		IF Trips_DB.Section[j].Sust.ChrgRly1FaultDelay_TON.Q = TRUE THEN 
			Trips_DB.Section[j].Sust.ChargeRelay1_FailtoClose := TRUE; 
			Trips_DB.Section[j].Sust.ChrgRly1FaultDelay_TON (IN:= FALSE);
		END_IF;
	ELSE
		Trips_DB.Section[j].Sust.ChrgRly1FaultDelay_TON (IN:= FALSE);	
	END_IF;

		//fail to open
	IF LCP.Section[j].Sust.CloseChargeRelay1 = FALSE AND LCP.Section[j].Sust.ChargeRelay1_close = TRUE THEN 
		//start timer
		Trips_DB.Section[j].Sust.ChrgRly1FaultDelay_TON (IN:= TRUE, PT := ChrgRlyFaultDelay_PT);
		
		IF Trips_DB.Section[j].Sust.ChrgRly1FaultDelay_TON.Q = TRUE THEN 
			Trips_DB.Section[j].Sust.ChargeRelay1_FailtoOpen := TRUE; 
			Trips_DB.Section[j].Sust.ChrgRly1FaultDelay_TON (IN:= FALSE);
		END_IF;
	ELSE
		Trips_DB.Section[j].Sust.ChrgRly1FaultDelay_TON (IN:= FALSE);
	END_IF;

	//Sust Charge rly2	
		//fail to close
	IF LCP.Section[j].Sust.CloseChargeRelay2 = TRUE AND LCP.Section[j].Sust.ChargeRelay2_close = FALSE THEN 
		//start timer
		Trips_DB.Section[j].Sust.ChrgRly2FaultDelay_TON (IN:= TRUE, PT := ChrgRlyFaultDelay_PT);
		
		IF Trips_DB.Section[j].Sust.ChrgRly2FaultDelay_TON.Q = TRUE THEN 
			Trips_DB.Section[j].Sust.ChargeRelay2_FailtoClose := TRUE;
			Trips_DB.Section[j].Sust.ChrgRly2FaultDelay_TON (IN:= FALSE);
		END_IF;
	ELSE
		Trips_DB.Section[j].Sust.ChrgRly2FaultDelay_TON (IN:= FALSE);
	END_IF;
	
		//fail to open
	IF LCP.Section[j].Sust.CloseChargeRelay2 = FALSE AND LCP.Section[j].Sust.ChargeRelay2_close = TRUE THEN 
		//start timer
		Trips_DB.Section[j].Sust.ChrgRly2FaultDelay_TON (IN:= TRUE, PT := ChrgRlyFaultDelay_PT);
		
		IF Trips_DB.Section[j].Sust.ChrgRly2FaultDelay_TON.Q = TRUE THEN 
			Trips_DB.Section[j].Sust.ChargeRelay2_FailtoOpen := TRUE; 
			Trips_DB.Section[j].Sust.ChrgRly2FaultDelay_TON (IN:= FALSE);
		END_IF;
	ELSE
		Trips_DB.Section[j].Sust.ChrgRly2FaultDelay_TON (IN:= FALSE);
	END_IF;

	//Sust dump rly1
		//fail to open
	IF LCP.Section[j].Sust.OpenDumpRelay1 = TRUE AND LCP.Section[j].Sust.DumpRelay1_close = TRUE THEN 
		//start timer
		Trips_DB.Section[j].Sust.DumpRly1FaultDelay_TON (IN := TRUE, PT := DumpRlyFaultDelay_PT);

		IF Trips_DB.Section[j].Sust.DumpRly1FaultDelay_TON.Q = TRUE THEN 
			Trips_DB.Section[j].Sust.DumpRelay1_FailtoOpen := TRUE; 
			Trips_DB.Section[j].Sust.DumpRly1FaultDelay_TON (IN:= FALSE);
		END_IF; 
	ELSE
		Trips_DB.Section[j].Sust.DumpRly1FaultDelay_TON (IN:= FALSE);
	END_IF;

		//fail to close
	IF LCP.Section[j].Sust.OpenDumpRelay1 = FALSE AND LCP.Section[j].Sust.DumpRelay1_close = FALSE THEN 
		//start timer
		Trips_DB.Section[j].Sust.DumpRly1FaultDelay_TON (IN := TRUE, PT := DumpRlyFaultDelay_PT); 
		
		IF Trips_DB.Section[j].Sust.DumpRly1FaultDelay_TON.Q = TRUE THEN 
			Trips_DB.Section[j].Sust.DumpRelay1_FailtoClose := TRUE; 
			Trips_DB.Section[j].Sust.DumpRly1FaultDelay_TON (IN:= FALSE);
		END_IF;
	ELSE
		Trips_DB.Section[j].Sust.DumpRly1FaultDelay_TON (IN:= FALSE);
	END_IF;

	//Sust dump rly2
		//fail to open
	IF LCP.Section[j].Sust.OpenDumpRelay2 = TRUE AND LCP.Section[j].Sust.DumpRelay2_close = TRUE THEN 
		//start timer
		Trips_DB.Section[j].Sust.DumpRly2FaultDelay_TON (IN := TRUE, PT := DumpRlyFaultDelay_PT); 
		
		IF Trips_DB.Section[j].Sust.DumpRly2FaultDelay_TON.Q = TRUE THEN 
			Trips_DB.Section[j].Sust.DumpRelay2_FailtoOpen := TRUE; 
			Trips_DB.Section[j].Sust.DumpRly2FaultDelay_TON (IN:= FALSE);
		END_IF;
	ELSE
		Trips_DB.Section[j].Sust.DumpRly2FaultDelay_TON (IN:= FALSE);
	END_IF;

		//fail to close
	IF LCP.Section[j].Sust.OpenDumpRelay2 = FALSE AND LCP.Section[j].Sust.DumpRelay2_close = FALSE THEN 
		//start timer
		Trips_DB.Section[j].Sust.DumpRly2FaultDelay_TON (IN := TRUE, PT := DumpRlyFaultDelay_PT); 
		IF Trips_DB.Section[j].Sust.DumpRly2FaultDelay_TON.Q = TRUE THEN 
			Trips_DB.Section[j].Sust.DumpRelay2_FailtoClose := TRUE; 
			Trips_DB.Section[j].Sust.DumpRly2FaultDelay_TON (IN:= FALSE);
		END_IF;
	ELSE
		Trips_DB.Section[j].Sust.DumpRly2FaultDelay_TON (IN:= FALSE);
	END_IF;
	
END_FOR;
//****************************************	
	
//Form Charge rly1
		//fail to close
IF LCP.Section[4].Form.CloseChargeRelay1 = TRUE AND LCP.Section[4].Form.ChargeRelay1_close = FALSE THEN 
		//start timer
		Trips_DB.Section[4].Form.ChrgRly1FaultDelay_TON (IN:= TRUE, PT := ChrgRlyFaultDelay_PT);
		
		IF Trips_DB.Section[4].Form.ChrgRly1FaultDelay_TON.Q = TRUE THEN 
			Trips_DB.Section[4].Form.ChargeRelay1_FailtoClose := TRUE; 
			Trips_DB.Section[4].Form.ChrgRly1FaultDelay_TON (IN:= FALSE);
		END_IF;
	ELSE
		Trips_DB.Section[4].Form.ChrgRly1FaultDelay_TON (IN:= FALSE);		
END_IF;

		//fail to open
IF LCP.Section[4].Form.CloseChargeRelay1 = FALSE AND LCP.Section[4].Form.ChargeRelay1_close = TRUE THEN 
		//start timer
		Trips_DB.Section[4].Form.ChrgRly1FaultDelay_TON (IN:= TRUE, PT := ChrgRlyFaultDelay_PT);
		
		IF Trips_DB.Section[4].Form.ChrgRly1FaultDelay_TON.Q = TRUE THEN 
			Trips_DB.Section[4].Form.ChargeRelay1_FailtoOpen := TRUE; 
			Trips_DB.Section[4].Form.ChrgRly1FaultDelay_TON (IN:= FALSE);
		END_IF;
	ELSE
		Trips_DB.Section[4].Form.ChrgRly1FaultDelay_TON (IN:= FALSE);
END_IF;

	//Form Charge rly2	
		//fail to close
IF LCP.Section[4].Form.CloseChargeRelay2 = TRUE AND LCP.Section[4].Form.ChargeRelay2_close = FALSE THEN 
		//start timer
		Trips_DB.Section[4].Form.ChrgRly2FaultDelay_TON (IN:= TRUE, PT := ChrgRlyFaultDelay_PT);
		
		IF Trips_DB.Section[4].Form.ChrgRly2FaultDelay_TON.Q = TRUE THEN 
			Trips_DB.Section[4].Form.ChargeRelay2_FailtoClose := TRUE; 
			Trips_DB.Section[4].Form.ChrgRly2FaultDelay_TON (IN:= FALSE);
		END_IF;
	ELSE
		Trips_DB.Section[4].Form.ChrgRly2FaultDelay_TON (IN:= FALSE);
END_IF;
	
		//fail to open
IF LCP.Section[4].Form.CloseChargeRelay2 = FALSE AND LCP.Section[4].Form.ChargeRelay2_close = TRUE THEN 
		//start timer
		Trips_DB.Section[4].Form.ChrgRly2FaultDelay_TON (IN:= TRUE, PT := ChrgRlyFaultDelay_PT);
		
		IF Trips_DB.Section[4].Form.ChrgRly2FaultDelay_TON.Q = TRUE THEN 
			Trips_DB.Section[4].Form.ChargeRelay2_FailtoOpen := TRUE; 
			Trips_DB.Section[4].Form.ChrgRly2FaultDelay_TON (IN:= FALSE);
		END_IF;
	ELSE
		Trips_DB.Section[4].Form.ChrgRly2FaultDelay_TON (IN:= FALSE);
END_IF;

	//Form dump rly1
		//fail to open
IF LCP.Section[4].Form.OpenDumpRelay1 = TRUE AND LCP.Section[4].Form.DumpRelay1_close = TRUE THEN 
		//start timer
		Trips_DB.Section[4].Form.DumpRly1FaultDelay_TON (IN := TRUE, PT := DumpRlyFaultDelay_PT);

		IF Trips_DB.Section[4].Form.DumpRly1FaultDelay_TON.Q = TRUE THEN 
			Trips_DB.Section[4].Form.DumpRelay1_FailtoOpen := TRUE; 
			Trips_DB.Section[4].Form.DumpRly1FaultDelay_TON (IN:= FALSE);
		END_IF; 
	ELSE
		Trips_DB.Section[4].Form.DumpRly1FaultDelay_TON (IN:= FALSE);
END_IF;

		//fail to close
IF LCP.Section[4].Form.OpenDumpRelay1 = FALSE AND LCP.Section[4].Form.DumpRelay1_close = FALSE THEN 
		//start timer
		Trips_DB.Section[4].Form.DumpRly1FaultDelay_TON (IN := TRUE, PT := DumpRlyFaultDelay_PT); 
		
		IF Trips_DB.Section[4].Form.DumpRly1FaultDelay_TON.Q = TRUE THEN 
			Trips_DB.Section[4].Form.DumpRelay1_FailtoClose := TRUE; 
			Trips_DB.Section[4].Form.DumpRly1FaultDelay_TON (IN:= FALSE);
		END_IF;
	ELSE
		Trips_DB.Section[4].Form.DumpRly1FaultDelay_TON (IN:= FALSE);
END_IF;

	//Form dump rly2
		//fail to open
IF LCP.Section[4].Form.OpenDumpRelay2 = TRUE AND LCP.Section[4].Form.DumpRelay2_close = TRUE THEN 
		//start timer
		Trips_DB.Section[4].Form.DumpRly2FaultDelay_TON (IN := TRUE, PT := DumpRlyFaultDelay_PT); 
		
		IF Trips_DB.Section[4].Form.DumpRly2FaultDelay_TON.Q = TRUE THEN 
			Trips_DB.Section[4].Form.DumpRelay2_FailtoOpen := TRUE; 
			Trips_DB.Section[4].Form.DumpRly2FaultDelay_TON (IN:= FALSE);
		END_IF;
	ELSE
		Trips_DB.Section[4].Form.DumpRly2FaultDelay_TON (IN:= FALSE);
END_IF;

		//fail to close
IF LCP.Section[4].Form.OpenDumpRelay2 = FALSE AND LCP.Section[4].Form.DumpRelay2_close = FALSE THEN 
		//start timer
		Trips_DB.Section[4].Form.DumpRly2FaultDelay_TON (IN := TRUE, PT := DumpRlyFaultDelay_PT); 
		IF Trips_DB.Section[4].Form.DumpRly2FaultDelay_TON.Q = TRUE THEN 
			Trips_DB.Section[4].Form.DumpRelay2_FailtoClose := TRUE; 
			Trips_DB.Section[4].Form.DumpRly2FaultDelay_TON (IN:= FALSE);
		END_IF;
	ELSE
		Trips_DB.Section[4].Form.DumpRly2FaultDelay_TON (IN:= FALSE);
END_IF;	

	//PreForm Charge rly
		//fail to close
IF (LCP.Section[4].Form.ClosePreFormChargeRly = TRUE AND LCP.Section[4].Form.PreFormChargeRly_close = FALSE) OR 
		(LCP.Section[4].Form.ClosePreFormChargeRly = FALSE AND LCP.Section[4].Form.PreFormChargeRly_close = TRUE) 
		THEN 
		//start timer
		Trips_DB.Section[4].Form.PreFormChrgRlyFaultDelay_TON (IN:= TRUE, PT := ChrgRlyFaultDelay_PT);
		
		IF Trips_DB.Section[4].Form.PreFormChrgRlyFaultDelay_TON.Q = TRUE THEN 
			Trips_DB.Section[4].Form.PreFormChrgRlyFailed := TRUE; 
			Trips_DB.Section[4].Form.PreFormChrgRlyFaultDelay_TON (IN:= FALSE);
		END_IF;
	ELSE
		Trips_DB.Section[4].Form.PreFormChrgRlyFaultDelay_TON (IN:= FALSE);
END_IF;

//form trigger charge 
		//fail to close
IF (LCP.Section[4].Form.CloseFormTrigChargeRly = TRUE AND LCP.Section[4].Form.FormTrigChargeRly_close = FALSE) OR 
		(LCP.Section[4].Form.CloseFormTrigChargeRly = FALSE AND LCP.Section[4].Form.FormTrigChargeRly_close = TRUE) 
		THEN 
		//start timer
		Trips_DB.Section[4].Form.FormTrigChrgRlyFaultDelay_TON (IN:= TRUE, PT := ChrgRlyFaultDelay_PT);
		
		IF Trips_DB.Section[4].Form.FormTrigChrgRlyFaultDelay_TON.Q = TRUE THEN 
			Trips_DB.Section[4].Form.FormTrigChrgRlyFailed := TRUE; 
			Trips_DB.Section[4].Form.FormTrigChrgRlyFaultDelay_TON (IN:= FALSE);
		END_IF;
	ELSE
		Trips_DB.Section[4].Form.FormTrigChrgRlyFaultDelay_TON (IN:= FALSE);
END_IF;

//preform trigger charge
		//fail to close
IF (LCP.Section[4].Form.ClosePreFormTrigChargeRly = TRUE AND LCP.Section[4].Form.PreFormTrigChargeRly_close = FALSE) OR 
		(LCP.Section[4].Form.ClosePreFormTrigChargeRly = FALSE AND LCP.Section[4].Form.PreFormTrigChargeRly_close = TRUE) 
		THEN 
		//start timer
		Trips_DB.Section[4].Form.PreFormTrigChrgRlyFaultDelay_TON (IN:= TRUE, PT := ChrgRlyFaultDelay_PT);
		
		IF Trips_DB.Section[4].Form.PreFormTrigChrgRlyFaultDelay_TON.Q = TRUE THEN 
			Trips_DB.Section[4].Form.PreFormTrigChrgRlyFailed := TRUE; 
			Trips_DB.Section[4].Form.PreFormTrigChrgRlyFaultDelay_TON (IN:= FALSE);
		END_IF;
	ELSE
		Trips_DB.Section[4].Form.PreFormTrigChrgRlyFaultDelay_TON (IN:= FALSE);
END_IF;

//preform dump
	//fail to close
IF (LCP.Section[4].Form.OpenPreFormDumpRly = TRUE AND LCP.Section[4].Form.PreFormDumpRly_close = FALSE) OR 
		(LCP.Section[4].Form.OpenPreFormDumpRly = FALSE AND LCP.Section[4].Form.PreFormDumpRly_close = TRUE) 
		THEN 
		//start timer
		Trips_DB.Section[4].Form.PreFormDumpRlyFaultDelay_TON (IN:= TRUE, PT := DumpRlyFaultDelay_PT);
		
		IF Trips_DB.Section[4].Form.PreFormDumpRlyFaultDelay_TON.Q = TRUE THEN 
			Trips_DB.Section[4].Form.PreFormDumpRlyFailed := TRUE; 
			Trips_DB.Section[4].Form.PreFormDumpRlyFaultDelay_TON (IN:= FALSE);
		END_IF;
	ELSE
		Trips_DB.Section[4].Form.PreFormDumpRlyFaultDelay_TON (IN:= FALSE);
END_IF;

//form trigger dump
	//fail to close
IF (LCP.Section[4].Form.OpenFormTrigDumpRly1 = TRUE AND LCP.Section[4].Form.FormTrigDumpRly1_close = FALSE) OR 
		(LCP.Section[4].Form.OpenFormTrigDumpRly1 = FALSE AND LCP.Section[4].Form.FormTrigDumpRly1_close = TRUE) 
		THEN 
		//start timer
		Trips_DB.Section[4].Form.FormTrigDumpRlyFaultDelay_TON (IN:= TRUE, PT := DumpRlyFaultDelay_PT);
		
		IF Trips_DB.Section[4].Form.FormTrigDumpRlyFaultDelay_TON.Q = TRUE THEN 
			Trips_DB.Section[4].Form.FormTrigDumpRly1Failed := TRUE; 
			Trips_DB.Section[4].Form.FormTrigDumpRlyFaultDelay_TON (IN:= FALSE);
		END_IF;
	ELSE
		Trips_DB.Section[4].Form.FormTrigDumpRlyFaultDelay_TON (IN:= FALSE);
END_IF;
	
//preform trigger dump
	//fail to close
IF (LCP.Section[4].Form.OpenPreFormTrigDumpRly1 = TRUE AND LCP.Section[4].Form.PreFormTrigDumpRly1_close = FALSE) OR 
		(LCP.Section[4].Form.OpenPreFormTrigDumpRly1 = FALSE AND LCP.Section[4].Form.PreFormTrigDumpRly1_close = TRUE) 
		THEN 
		//start timer
		Trips_DB.Section[4].Form.PreFormTrigDumpRlyFaultDelay_TON (IN:= TRUE, PT := DumpRlyFaultDelay_PT);
		
		IF Trips_DB.Section[4].Form.PreFormTrigDumpRlyFaultDelay_TON.Q = TRUE THEN 
			Trips_DB.Section[4].Form.PreFormTrigDumpRly1Failed := TRUE; 
			Trips_DB.Section[4].Form.PreFormTrigDumpRlyFaultDelay_TON (IN:= FALSE);
		END_IF;
	ELSE
		Trips_DB.Section[4].Form.PreFormTrigDumpRlyFaultDelay_TON (IN:= FALSE);
END_IF;
	

// if rly fail to close or fail to open then trips_db.rly_failed - for alarms	
FOR j := 1 TO 3 BY 1 DO
	//peak
	IF Trips_DB.Section[j].Peak.ChargeRelay1_FailtoClose = TRUE OR Trips_DB.Section[j].Peak.ChargeRelay1_FailtoOpen = TRUE THEN
		Trips_DB.Section[j].Peak.ChargeRelay1_Failed := TRUE;  
	END_IF;
	
	IF Trips_DB.Section[j].Peak.ChargeRelay2_FailtoClose = TRUE OR Trips_DB.Section[j].Peak.ChargeRelay2_FailtoOpen = TRUE THEN
		Trips_DB.Section[j].Peak.ChargeRelay2_Failed := TRUE;  
	END_IF;
	
	IF Trips_DB.Section[j].Peak.DumpRelay1_FailtoClose = TRUE OR Trips_DB.Section[j].Peak.DumpRelay1_FailtoOpen = TRUE THEN
		Trips_DB.Section[j].Peak.DumpRelay1_Failed := TRUE;  
	END_IF;
	
	IF Trips_DB.Section[j].Peak.DumpRelay2_FailtoClose = TRUE OR Trips_DB.Section[j].Peak.DumpRelay2_FailtoOpen = TRUE THEN
		Trips_DB.Section[j].Peak.DumpRelay2_Failed := TRUE;  
	END_IF;
	
	//sust
	IF Trips_DB.Section[j].Sust.ChargeRelay1_FailtoClose = TRUE OR Trips_DB.Section[j].Sust.ChargeRelay1_FailtoOpen = TRUE THEN
		Trips_DB.Section[j].Sust.ChargeRelay1_Failed := TRUE;  
	END_IF;
	
	IF Trips_DB.Section[j].Sust.ChargeRelay2_FailtoClose = TRUE OR Trips_DB.Section[j].Sust.ChargeRelay2_FailtoOpen = TRUE THEN
		Trips_DB.Section[j].Sust.ChargeRelay2_Failed := TRUE;  
	END_IF;
	
	IF Trips_DB.Section[j].Sust.DumpRelay1_FailtoClose = TRUE OR Trips_DB.Section[j].Sust.DumpRelay1_FailtoOpen = TRUE THEN
		Trips_DB.Section[j].Sust.DumpRelay1_Failed := TRUE;  
	END_IF;
	
	IF Trips_DB.Section[j].Sust.DumpRelay2_FailtoClose = TRUE OR Trips_DB.Section[j].Sust.DumpRelay2_FailtoOpen = TRUE THEN
		Trips_DB.Section[j].Sust.DumpRelay2_Failed := TRUE;  
	END_IF;
	
END_FOR;

//any system tripped
FOR k := 1 TO 4 BY 1 DO
	IF Trips_DB.Section[k].SystemTripped = TRUE OR Trips_DB.MCPsystemTripped = TRUE THEN
		Trips_DB.AnySystemTripped := TRUE;
		ELSE
			Trips_DB.AnySystemTripped := FALSE;
	END_IF;
END_FOR

// no faulted detected
IF (Trips_DB.AnySystemTripped = FALSE AND
	Trips_DB.AnyChargerOverTemp = FALSE AND
	Trips_DB.AnyChargerLoadFault = FALSE AND  //no charger fault is a permissives to charge
	Trips_DB.AnyChargerInterlockOpen = FALSE AND
	Trips_DB.AnyChargerFaulted = FALSE AND
	Trips_DB.AnyEstopPressed = FALSE AND
	Trips_DB.AnyDumpRlyFail = FALSE AND
	Trips_DB.AnyChargeRlyFail = FALSE AND 
	Trips_DB.AllDCpsuOK = TRUE AND
	Trips_DB.AnyLossInhibitSignal = FALSE AND
	Trips_DB.AnyLossHVONsignal = FALSE AND 
	Trips_DB.MachineGNDrlyFailed = FALSE AND 
	Trips_DB.ChargingTimerRunout = FALSE AND
	Trips_DB.ChargedTimerRunout = FALSE AND
	Trips_DB.DumpTimerRunout) OR HMI_DB.NoFaultDetectedBP = TRUE //admin bypass
	THEN
		Trips_DB.NoFaultDetected := TRUE;
	ELSE
		Trips_DB.NoFaultDetected := FALSE;
END_IF;


(*
FOR i := 1 TO 10 BY 1 DO
	IF (Trips_DB.Coil[i].ACInterlockRelayFailedtoClose = TRUE OR 
		Trips_DB.Coil[i].ACInterlockRelayFailedtoOpen = TRUE OR 
		Trips_DB.Coil[i].ChargeRelay_FailtoClose = TRUE OR
		Trips_DB.Coil[i].ChargeRelay_FailtoOpen = TRUE OR
		Trips_DB.Coil[i].DumpRelay1_FailtoClose =  TRUE OR 
		Trips_DB.Coil[i].DumpRelay1_FailtoOpen = TRUE OR 
		Trips_DB.Coil[i].DumpRelay2_FailtoClose =  TRUE OR 
		Trips_DB.Coil[i].DumpRelay2_FailtoOpen = TRUE OR 
		Trips_DB.Coil[i].ChargerVoltageReadingFaulted = TRUE OR
		Trips_DB.Coil[i].CurrentReadingFaulted = TRUE OR
		Devices.Coil[i].Local_EstopPB_Pressed = TRUE OR
		Devices.Coil[i].LossPneumaticPressure = FALSE) AND Devices.Coil[i].CoilEnabled = TRUE 	
		THEN
			Devices.Coil[i].SystemFaulted := TRUE;
	END_IF
	
	IF Devices.Coil[i].SystemFaulted = TRUE THEN
		Trips_DB.SystemTripped := TRUE;
	END_IF;
END_FOR;

//*********************************** Test
(*IF InstrumentReading.R2_01_CH01 <= 0.0 THEN
	delay2s(input := FALSE);
ELSE 
	delay2s (input := TRUE);
END_IF;
bTest := delay2s.output;
*)
// Instrumentation Hardware trip
//Input.R2_01_00_Status.0;
*)
//************** Clear System Fault
IF Trips_DB.ClearAllFaults = TRUE OR stControl.ClearAllFaults = TRUE THEN
	//Trips_DB.InstrumentationFaulted := FALSE;

	Trips_DB.MCPsystemTripped := FALSE; //reset mcp trip
	Trips_DB.AnyChargerOverTemp := FALSE;
	Trips_DB.AnyChargerLoadFault := FALSE;  
	Trips_DB.AnyChargerInterlockOpen := FALSE;
	Trips_DB.AnyChargerFaulted := FALSE;
	Trips_DB.AnyEstopPressed := FALSE;
	Trips_DB.AnyDumpRlyFail := FALSE;
	Trips_DB.AnyChargeRlyFail := FALSE;
	Trips_DB.MasterStopPBPressed := FALSE; //this is only for alarms
	Trips_DB.CageEStopCircuitBroken := FALSE;
	Trips_DB.MCPLossDCpower := FALSE;
	Trips_DB.AnyLossInhibitSignal := FALSE;
	Trips_DB.AnyLossHVONsignal := FALSE;
	Trips_DB.MachineGNDrlyFailed := FALSE;
	Trips_DB.ChargingTimerRunout := FALSE;
	Trips_DB.ChargedTimerRunout  := FALSE;
	Trips_DB.DumpTimerRunout := FALSE;
	//Trips_DB.AnyACInterlockFail := FALSE;
	//reset relay trips
	FOR j := 1 TO 3 BY 1 DO 
		//reset relay faults
		Trips_DB.Section[j].SystemTripped := FALSE;
		//Peaking
		Trips_DB.Section[j].Peak.DumpRelay1_FailtoClose := FALSE;
		Trips_DB.Section[j].Peak.DumpRelay1_FailtoOpen := FALSE;
		Trips_DB.Section[j].Peak.DumpRelay2_FailtoClose := FALSE;
		Trips_DB.Section[j].Peak.DumpRelay2_FailtoOpen := FALSE;
		Trips_DB.Section[j].Peak.ChargeRelay1_FailtoClose := FALSE;
		Trips_DB.Section[j].Peak.ChargeRelay1_FailtoOpen := FALSE;
		Trips_DB.Section[j].Peak.ChargeRelay2_FailtoClose := FALSE;
		Trips_DB.Section[j].Peak.ChargeRelay2_FailtoOpen := FALSE;
		//Sust
		Trips_DB.Section[j].Sust.DumpRelay1_FailtoClose := FALSE;
		Trips_DB.Section[j].Sust.DumpRelay1_FailtoOpen := FALSE;
		Trips_DB.Section[j].Sust.DumpRelay2_FailtoClose := FALSE;
		Trips_DB.Section[j].Sust.DumpRelay2_FailtoOpen := FALSE;
		Trips_DB.Section[j].Sust.ChargeRelay1_FailtoClose := FALSE;
		Trips_DB.Section[j].Sust.ChargeRelay1_FailtoOpen := FALSE;
		Trips_DB.Section[j].Sust.ChargeRelay2_FailtoClose := FALSE;
		Trips_DB.Section[j].Sust.ChargeRelay2_FailtoOpen := FALSE;
	
	END_FOR;
	
	//FORM
	Trips_DB.Section[4].Form.ChargeRelay1_FailtoOpen := FALSE;
	Trips_DB.Section[4].Form.ChargeRelay1_FailtoClose := FALSE;
	Trips_DB.Section[4].Form.ChargeRelay1_Failed:= FALSE;
	Trips_DB.Section[4].Form.ChargeRelay2_FailtoOpen := FALSE;
	Trips_DB.Section[4].Form.ChargeRelay2_FailtoClose := FALSE;
	Trips_DB.Section[4].Form.ChargeRelay2_Failed:= FALSE;
	
	Trips_DB.Section[4].Form.DumpRelay1_FailtoOpen := FALSE;
	Trips_DB.Section[4].Form.DumpRelay1_FailtoClose := FALSE;
	Trips_DB.Section[4].Form.DumpRelay1_Failed := FALSE;
	Trips_DB.Section[4].Form.DumpRelay2_FailtoOpen := FALSE;
	Trips_DB.Section[4].Form.DumpRelay2_FailtoClose := FALSE;
	Trips_DB.Section[4].Form.DumpRelay2_Failed := FALSE;
	
	Trips_DB.Section[4].Form.PreFormChrgRlyFailed := FALSE;
	Trips_DB.Section[4].Form.FormTrigChrgRlyFailed := FALSE;
	Trips_DB.Section[4].Form.PreFormTrigChrgRlyFailed := FALSE;
	Trips_DB.Section[4].Form.PreFormDumpRlyFailed := FALSE;
	Trips_DB.Section[4].Form.FormTrigDumpRly1Failed := FALSE;
	Trips_DB.Section[4].Form.PreFormTrigDumpRly1Failed := FALSE;
	
	Trips_DB.Section[4].SystemTripped := FALSE;
	
	evtLogger.ClearAllAlarms(0, FALSE);
	//evtLogger.ClearLoggedEvents(1);
END_IF;


IF i > 8 THEN 
	i := 1;
END_IF;

IF j > 3 THEN 
	j := 1;
END_IF;

IF k > 4 THEN 
	k := 1;
END_IF;

END_PROGRAM

// ---- POUs/Alarms.TcPOU
PROGRAM Alarms
VAR
	bWarning : BOOL;
	bConfirm : BOOL;
	alarms : ARRAY[0..431] OF Alarms_FB;
	
END_VAR

// Alarm Word 1 - MCP Alarms
//MCP Alarms

Alarms_DB.MCP.AlarmWord.0 := Trips_DB.MasterStopPBPressed;
Alarms_DB.MCP.AlarmWord.1 := Trips_DB.CageEStopCircuitBroken;
Alarms_DB.MCP.AlarmWord.2 := Trips_DB.LocalModeSelected;
Alarms_DB.MCP.AlarmWord.3 := Trips_DB.MCPLossDCpower;
Alarms_DB.MCP.AlarmWord.4 := MCP_IO.Charger[1].SummaryFaulted;
Alarms_DB.MCP.AlarmWord.5 := MCP_IO.Charger[2].SummaryFaulted;
Alarms_DB.MCP.AlarmWord.6 := MCP_IO.Charger[3].SummaryFaulted;
Alarms_DB.MCP.AlarmWord.7 := MCP_IO.Charger[4].SummaryFaulted;
Alarms_DB.MCP.AlarmWord.8 := MCP_IO.Charger[5].SummaryFaulted;
Alarms_DB.MCP.AlarmWord.9 := MCP_IO.Charger[6].SummaryFaulted;
Alarms_DB.MCP.AlarmWord.10 := MCP_IO.Charger[7].SummaryFaulted;
Alarms_DB.MCP.AlarmWord.11 := MCP_IO.Charger[8].SummaryFaulted;
Alarms_DB.MCP.AlarmWord.12 := Trips_DB.ChargedTimerRunout;
Alarms_DB.MCP.AlarmWord.13 := Trips_DB.ChargingTimerRunout;
Alarms_DB.MCP.AlarmWord.14 := Trips_DB.MCPsystemTripped;
Alarms_DB.MCP.AlarmWord.15 := Trips_DB.AnyEstopPressed;

//Alarm Word 1 msg
//IE: alarms[299](evtEntry:= Tc_Events.AlarmWord11.b4, bEvt:= gvl.test, bConfirm:= bConfirm);
alarms[0](evtEntry:= Tc_Events.AlarmWord1.b0, bEvt:= Alarms_DB.MCP.AlarmWord.0, bConfirm:= bConfirm);
alarms[1](evtEntry:= Tc_Events.AlarmWord1.b1, bEvt:= Alarms_DB.MCP.AlarmWord.1, bConfirm:= bConfirm);
alarms[2](evtEntry:= Tc_Events.AlarmWord1.b2, bEvt:= Alarms_DB.MCP.AlarmWord.2, bConfirm:= bConfirm);
alarms[3](evtEntry:= Tc_Events.AlarmWord1.b3, bEvt:= Alarms_DB.MCP.AlarmWord.3, bConfirm:= bConfirm);
alarms[4](evtEntry:= Tc_Events.AlarmWord1.b4, bEvt:= Alarms_DB.MCP.AlarmWord.4, bConfirm:= bConfirm);
alarms[5](evtEntry:= Tc_Events.AlarmWord1.b5, bEvt:= Alarms_DB.MCP.AlarmWord.5, bConfirm:= bConfirm);
alarms[6](evtEntry:= Tc_Events.AlarmWord1.b6, bEvt:= Alarms_DB.MCP.AlarmWord.6, bConfirm:= bConfirm);
alarms[7](evtEntry:= Tc_Events.AlarmWord1.b7, bEvt:= Alarms_DB.MCP.AlarmWord.7, bConfirm:= bConfirm);
alarms[8](evtEntry:= Tc_Events.AlarmWord1.b8, bEvt:= Alarms_DB.MCP.AlarmWord.8, bConfirm:= bConfirm);
alarms[9](evtEntry:= Tc_Events.AlarmWord1.b9, bEvt:= Alarms_DB.MCP.AlarmWord.9, bConfirm:= bConfirm);
alarms[0](evtEntry:= Tc_Events.AlarmWord1.b10, bEvt:= Alarms_DB.MCP.AlarmWord.10, bConfirm:= bConfirm);
alarms[11](evtEntry:= Tc_Events.AlarmWord1.b11, bEvt:= Alarms_DB.MCP.AlarmWord.11, bConfirm:= bConfirm);
alarms[12](evtEntry:= Tc_Events.AlarmWord1.b12, bEvt:= Alarms_DB.MCP.AlarmWord.12, bConfirm:= bConfirm);
alarms[13](evtEntry:= Tc_Events.AlarmWord1.b13, bEvt:= Alarms_DB.MCP.AlarmWord.13, bConfirm:= bConfirm);
alarms[14](evtEntry:= Tc_Events.AlarmWord1.b14, bEvt:= Alarms_DB.MCP.AlarmWord.14, bConfirm:= bConfirm);
alarms[15](evtEntry:= Tc_Events.AlarmWord1.b15, bEvt:= Alarms_DB.MCP.AlarmWord.15, bConfirm:= bConfirm);

// Alarm Word 2 - Section 1 Alarms
Alarms_DB.Section1.AlarmWord.0 := Trips_DB.Section[1].SystemTripped;
Alarms_DB.Section1.AlarmWord.1 := Trips_DB.Section[1].LossPneumaticPressure;
Alarms_DB.Section1.AlarmWord.2 := Trips_DB.Section[1].Peak.ChargeRelay1_Failed;
Alarms_DB.Section1.AlarmWord.3 := Trips_DB.Section[1].Peak.ChargeRelay2_Failed;
Alarms_DB.Section1.AlarmWord.4 := Trips_DB.Section[1].Peak.DumpRelay1_Failed;
Alarms_DB.Section1.AlarmWord.5 := Trips_DB.Section[1].Peak.DumpRelay2_Failed;
Alarms_DB.Section1.AlarmWord.6 := Trips_DB.Section[1].Sust.ChargeRelay1_Failed;
Alarms_DB.Section1.AlarmWord.7 := Trips_DB.Section[1].Sust.ChargeRelay2_Failed;
Alarms_DB.Section1.AlarmWord.8 := Trips_DB.Section[1].Sust.DumpRelay1_Failed;
Alarms_DB.Section1.AlarmWord.9 := Trips_DB.Section[1].Sust.DumpRelay2_Failed;
Alarms_DB.Section1.AlarmWord.10 := Trips_DB.Section[1].LossDCPower;


// Alarm Word 2 - Msg
alarms[16](evtEntry:= Tc_Events.AlarmWord2.b0, bEvt:= Alarms_DB.Section1.AlarmWord.0, bConfirm:= bConfirm);
alarms[17](evtEntry:= Tc_Events.AlarmWord2.b1, bEvt:= Alarms_DB.Section1.AlarmWord.1, bConfirm:= bConfirm);
alarms[18](evtEntry:= Tc_Events.AlarmWord2.b2, bEvt:= Alarms_DB.Section1.AlarmWord.2, bConfirm:= bConfirm);
alarms[19](evtEntry:= Tc_Events.AlarmWord2.b3, bEvt:= Alarms_DB.Section1.AlarmWord.3, bConfirm:= bConfirm);
alarms[20](evtEntry:= Tc_Events.AlarmWord2.b4, bEvt:= Alarms_DB.Section1.AlarmWord.4, bConfirm:= bConfirm);
alarms[21](evtEntry:= Tc_Events.AlarmWord2.b5, bEvt:= Alarms_DB.Section1.AlarmWord.5, bConfirm:= bConfirm);
alarms[22](evtEntry:= Tc_Events.AlarmWord2.b6, bEvt:= Alarms_DB.Section1.AlarmWord.6, bConfirm:= bConfirm);
alarms[23](evtEntry:= Tc_Events.AlarmWord2.b7, bEvt:= Alarms_DB.Section1.AlarmWord.7, bConfirm:= bConfirm);
alarms[24](evtEntry:= Tc_Events.AlarmWord2.b8, bEvt:= Alarms_DB.Section1.AlarmWord.8, bConfirm:= bConfirm);
alarms[25](evtEntry:= Tc_Events.AlarmWord2.b9, bEvt:= Alarms_DB.Section1.AlarmWord.9, bConfirm:= bConfirm);
alarms[26](evtEntry:= Tc_Events.AlarmWord2.b10, bEvt:= Alarms_DB.Section1.AlarmWord.10, bConfirm:= bConfirm);
//alarms[27] - spare
//alarms[28] - spare
//alarms[29] - spare
//alarms[30] - spare
//alarms[31] - spare


// Alarm Word 3 - Section 2 Alarms
Alarms_DB.Section2.AlarmWord.0 := Trips_DB.Section[2].SystemTripped;
Alarms_DB.Section2.AlarmWord.1 := Trips_DB.Section[2].LossPneumaticPressure;
Alarms_DB.Section2.AlarmWord.2 := Trips_DB.Section[2].Peak.ChargeRelay1_Failed;
Alarms_DB.Section2.AlarmWord.3 := Trips_DB.Section[2].Peak.ChargeRelay2_Failed;
Alarms_DB.Section2.AlarmWord.4 := Trips_DB.Section[2].Peak.DumpRelay1_Failed;
Alarms_DB.Section2.AlarmWord.5 := Trips_DB.Section[2].Peak.DumpRelay2_Failed;
Alarms_DB.Section2.AlarmWord.6 := Trips_DB.Section[2].Sust.ChargeRelay1_Failed;
Alarms_DB.Section2.AlarmWord.7 := Trips_DB.Section[2].Sust.ChargeRelay2_Failed;
Alarms_DB.Section2.AlarmWord.8 := Trips_DB.Section[2].Sust.DumpRelay1_Failed;
Alarms_DB.Section2.AlarmWord.9 := Trips_DB.Section[2].Sust.DumpRelay2_Failed;
Alarms_DB.Section2.AlarmWord.10 := Trips_DB.Section[2].LossDCPower;


// Alarm Word 3 - Msg
alarms[32](evtEntry:= Tc_Events.AlarmWord3.b0, bEvt:= Alarms_DB.Section2.AlarmWord.0, bConfirm:= bConfirm);
alarms[33](evtEntry:= Tc_Events.AlarmWord3.b1, bEvt:= Alarms_DB.Section2.AlarmWord.1, bConfirm:= bConfirm);
alarms[34](evtEntry:= Tc_Events.AlarmWord3.b2, bEvt:= Alarms_DB.Section2.AlarmWord.2, bConfirm:= bConfirm);
alarms[35](evtEntry:= Tc_Events.AlarmWord3.b3, bEvt:= Alarms_DB.Section2.AlarmWord.3, bConfirm:= bConfirm);
alarms[36](evtEntry:= Tc_Events.AlarmWord3.b4, bEvt:= Alarms_DB.Section2.AlarmWord.4, bConfirm:= bConfirm);
alarms[37](evtEntry:= Tc_Events.AlarmWord3.b5, bEvt:= Alarms_DB.Section2.AlarmWord.5, bConfirm:= bConfirm);
alarms[38](evtEntry:= Tc_Events.AlarmWord3.b6, bEvt:= Alarms_DB.Section2.AlarmWord.6, bConfirm:= bConfirm);
alarms[39](evtEntry:= Tc_Events.AlarmWord3.b7, bEvt:= Alarms_DB.Section2.AlarmWord.7, bConfirm:= bConfirm);
alarms[40](evtEntry:= Tc_Events.AlarmWord3.b8, bEvt:= Alarms_DB.Section2.AlarmWord.8, bConfirm:= bConfirm);
alarms[41](evtEntry:= Tc_Events.AlarmWord3.b9, bEvt:= Alarms_DB.Section2.AlarmWord.9, bConfirm:= bConfirm);
alarms[42](evtEntry:= Tc_Events.AlarmWord3.b10, bEvt:= Alarms_DB.Section2.AlarmWord.10, bConfirm:= bConfirm);
//alarms[43] - spare
//alarms[44] - spare
//alarms[45] - spare
//alarms[46] - spare
//alarms[47] - spare

// Alarm Word 4 - Section 3 Alarms
Alarms_DB.Section3.AlarmWord.0 := Trips_DB.Section[3].SystemTripped;
Alarms_DB.Section3.AlarmWord.1 := Trips_DB.Section[3].LossPneumaticPressure;
Alarms_DB.Section3.AlarmWord.2 := Trips_DB.Section[3].Peak.ChargeRelay1_Failed;
Alarms_DB.Section3.AlarmWord.3 := Trips_DB.Section[3].Peak.ChargeRelay2_Failed;
Alarms_DB.Section3.AlarmWord.4 := Trips_DB.Section[3].Peak.DumpRelay1_Failed;
Alarms_DB.Section3.AlarmWord.5 := Trips_DB.Section[3].Peak.DumpRelay2_Failed;
Alarms_DB.Section3.AlarmWord.6 := Trips_DB.Section[3].Sust.ChargeRelay1_Failed;
Alarms_DB.Section3.AlarmWord.7 := Trips_DB.Section[3].Sust.ChargeRelay2_Failed;
Alarms_DB.Section3.AlarmWord.8 := Trips_DB.Section[3].Sust.DumpRelay1_Failed;
Alarms_DB.Section3.AlarmWord.9 := Trips_DB.Section[3].Sust.DumpRelay2_Failed;
Alarms_DB.Section3.AlarmWord.10 := Trips_DB.Section[3].LossDCPower;


// Alarm Word 4 - Msg
alarms[48](evtEntry:= Tc_Events.AlarmWord4.b0, bEvt:= Alarms_DB.Section3.AlarmWord.0, bConfirm:= bConfirm);
alarms[49](evtEntry:= Tc_Events.AlarmWord4.b1, bEvt:= Alarms_DB.Section3.AlarmWord.1, bConfirm:= bConfirm);
alarms[50](evtEntry:= Tc_Events.AlarmWord4.b2, bEvt:= Alarms_DB.Section3.AlarmWord.2, bConfirm:= bConfirm);
alarms[51](evtEntry:= Tc_Events.AlarmWord4.b3, bEvt:= Alarms_DB.Section3.AlarmWord.3, bConfirm:= bConfirm);
alarms[52](evtEntry:= Tc_Events.AlarmWord4.b4, bEvt:= Alarms_DB.Section3.AlarmWord.4, bConfirm:= bConfirm);
alarms[53](evtEntry:= Tc_Events.AlarmWord4.b5, bEvt:= Alarms_DB.Section3.AlarmWord.5, bConfirm:= bConfirm);
alarms[54](evtEntry:= Tc_Events.AlarmWord4.b6, bEvt:= Alarms_DB.Section3.AlarmWord.6, bConfirm:= bConfirm);
alarms[55](evtEntry:= Tc_Events.AlarmWord4.b7, bEvt:= Alarms_DB.Section3.AlarmWord.7, bConfirm:= bConfirm);
alarms[56](evtEntry:= Tc_Events.AlarmWord4.b8, bEvt:= Alarms_DB.Section3.AlarmWord.8, bConfirm:= bConfirm);
alarms[57](evtEntry:= Tc_Events.AlarmWord4.b9, bEvt:= Alarms_DB.Section3.AlarmWord.9, bConfirm:= bConfirm);
alarms[58](evtEntry:= Tc_Events.AlarmWord4.b10, bEvt:= Alarms_DB.Section3.AlarmWord.10, bConfirm:= bConfirm);
//alarms[59] - spare
//alarms[60] - spare
//alarms[61] - spare
//alarms[62] - spare
//alarms[63] - spare

// Alarm Word 5 - Section 4 Alarms
Alarms_DB.Section4.AlarmWord.0 := Trips_DB.Section[4].SystemTripped;
Alarms_DB.Section4.AlarmWord.1 := Trips_DB.Section[4].LossPneumaticPressure;
Alarms_DB.Section4.AlarmWord.2 := Trips_DB.Section[4].Form.ChargeRelay1_Failed;
Alarms_DB.Section4.AlarmWord.3 := Trips_DB.Section[4].Form.ChargeRelay2_Failed;
Alarms_DB.Section4.AlarmWord.4 := Trips_DB.Section[4].Form.DumpRelay1_Failed;
Alarms_DB.Section4.AlarmWord.5 := Trips_DB.Section[4].Form.DumpRelay2_Failed;
Alarms_DB.Section4.AlarmWord.6 := Trips_DB.Section[4].Form.PreFormChrgRlyFailed;
Alarms_DB.Section4.AlarmWord.7 := Trips_DB.Section[4].Form.FormTrigChrgRlyFailed;
Alarms_DB.Section4.AlarmWord.8 := Trips_DB.Section[4].Form.PreFormTrigChrgRlyFailed;
Alarms_DB.Section4.AlarmWord.9 := Trips_DB.Section[4].Form.PreFormDumpRlyFailed;
Alarms_DB.Section4.AlarmWord.10 := Trips_DB.Section[4].Form.FormTrigDumpRly1Failed;
Alarms_DB.Section4.AlarmWord.11 := Trips_DB.Section[4].Form.PreFormTrigDumpRly1Failed;
Alarms_DB.Section4.AlarmWord.12 := Trips_DB.Section[4].LossDCPower;

// Alarm Word 5 - Msg
alarms[64](evtEntry:= Tc_Events.AlarmWord5.b0, bEvt:= Alarms_DB.Section4.AlarmWord.0, bConfirm:= bConfirm);
alarms[65](evtEntry:= Tc_Events.AlarmWord5.b1, bEvt:= Alarms_DB.Section4.AlarmWord.1, bConfirm:= bConfirm);
alarms[66](evtEntry:= Tc_Events.AlarmWord5.b2, bEvt:= Alarms_DB.Section4.AlarmWord.2, bConfirm:= bConfirm);
alarms[67](evtEntry:= Tc_Events.AlarmWord5.b3, bEvt:= Alarms_DB.Section4.AlarmWord.3, bConfirm:= bConfirm);
alarms[68](evtEntry:= Tc_Events.AlarmWord5.b4, bEvt:= Alarms_DB.Section4.AlarmWord.4, bConfirm:= bConfirm);
alarms[69](evtEntry:= Tc_Events.AlarmWord5.b5, bEvt:= Alarms_DB.Section4.AlarmWord.5, bConfirm:= bConfirm);
alarms[70](evtEntry:= Tc_Events.AlarmWord5.b6, bEvt:= Alarms_DB.Section4.AlarmWord.6, bConfirm:= bConfirm);
alarms[71](evtEntry:= Tc_Events.AlarmWord5.b7, bEvt:= Alarms_DB.Section4.AlarmWord.7, bConfirm:= bConfirm);
alarms[72](evtEntry:= Tc_Events.AlarmWord5.b8, bEvt:= Alarms_DB.Section4.AlarmWord.8, bConfirm:= bConfirm);
alarms[73](evtEntry:= Tc_Events.AlarmWord5.b9, bEvt:= Alarms_DB.Section4.AlarmWord.9, bConfirm:= bConfirm);
alarms[74](evtEntry:= Tc_Events.AlarmWord5.b10, bEvt:= Alarms_DB.Section4.AlarmWord.10, bConfirm:= bConfirm);
alarms[75](evtEntry:= Tc_Events.AlarmWord5.b10, bEvt:= Alarms_DB.Section4.AlarmWord.11, bConfirm:= bConfirm);
alarms[76](evtEntry:= Tc_Events.AlarmWord5.b10, bEvt:= Alarms_DB.Section4.AlarmWord.12, bConfirm:= bConfirm);
//alarms[77] - spare
//alarms[78] - spare
//alarms[79] - spare

// Alarm Word 6 - Alarms
Alarms_DB.AlarmWord6.AlarmWord.0:= Trips_DB.Charger[1].OverTemp;
Alarms_DB.AlarmWord6.AlarmWord.1 := Trips_DB.Charger[1].InterlockOpen;
Alarms_DB.AlarmWord6.AlarmWord.2 := Trips_DB.Charger[1].LoadFaulted;
Alarms_DB.AlarmWord6.AlarmWord.3 := Trips_DB.Charger[2].OverTemp;
Alarms_DB.AlarmWord6.AlarmWord.4 := Trips_DB.Charger[2].InterlockOpen;
Alarms_DB.AlarmWord6.AlarmWord.5 := Trips_DB.Charger[2].LoadFaulted;
Alarms_DB.AlarmWord6.AlarmWord.6 := Trips_DB.Charger[3].OverTemp;
Alarms_DB.AlarmWord6.AlarmWord.7 := Trips_DB.Charger[3].InterlockOpen;
Alarms_DB.AlarmWord6.AlarmWord.8 := Trips_DB.Charger[3].LoadFaulted;
Alarms_DB.AlarmWord6.AlarmWord.9 := Trips_DB.Charger[4].OverTemp;
Alarms_DB.AlarmWord6.AlarmWord.10 := Trips_DB.Charger[4].InterlockOpen;
Alarms_DB.AlarmWord6.AlarmWord.11 := Trips_DB.Charger[4].LoadFaulted;
Alarms_DB.AlarmWord6.AlarmWord.12 := Trips_DB.Charger[5].OverTemp;
Alarms_DB.AlarmWord6.AlarmWord.13 := Trips_DB.Charger[5].InterlockOpen;
Alarms_DB.AlarmWord6.AlarmWord.14 := Trips_DB.Charger[5].LoadFaulted;

// Alarm Word 6 - Msg
alarms[80](evtEntry:= Tc_Events.AlarmWord6.b0, bEvt:= Alarms_DB.AlarmWord6.AlarmWord.0, bConfirm:= bConfirm);
alarms[81](evtEntry:= Tc_Events.AlarmWord6.b1, bEvt:= Alarms_DB.AlarmWord6.AlarmWord.1, bConfirm:= bConfirm);
alarms[82](evtEntry:= Tc_Events.AlarmWord6.b2, bEvt:= Alarms_DB.AlarmWord6.AlarmWord.2, bConfirm:= bConfirm);
alarms[83](evtEntry:= Tc_Events.AlarmWord6.b3, bEvt:= Alarms_DB.AlarmWord6.AlarmWord.3, bConfirm:= bConfirm);
alarms[84](evtEntry:= Tc_Events.AlarmWord6.b4, bEvt:= Alarms_DB.AlarmWord6.AlarmWord.4, bConfirm:= bConfirm);
alarms[85](evtEntry:= Tc_Events.AlarmWord6.b5, bEvt:= Alarms_DB.AlarmWord6.AlarmWord.5, bConfirm:= bConfirm);
alarms[86](evtEntry:= Tc_Events.AlarmWord6.b6, bEvt:= Alarms_DB.AlarmWord6.AlarmWord.6, bConfirm:= bConfirm);
alarms[87](evtEntry:= Tc_Events.AlarmWord6.b7, bEvt:= Alarms_DB.AlarmWord6.AlarmWord.7, bConfirm:= bConfirm);
alarms[88](evtEntry:= Tc_Events.AlarmWord6.b8, bEvt:= Alarms_DB.AlarmWord6.AlarmWord.8, bConfirm:= bConfirm);
alarms[89](evtEntry:= Tc_Events.AlarmWord6.b9, bEvt:= Alarms_DB.AlarmWord6.AlarmWord.9, bConfirm:= bConfirm);
alarms[90](evtEntry:= Tc_Events.AlarmWord6.b10, bEvt:= Alarms_DB.AlarmWord6.AlarmWord.10, bConfirm:= bConfirm);
alarms[91](evtEntry:= Tc_Events.AlarmWord6.b11, bEvt:= Alarms_DB.AlarmWord6.AlarmWord.11, bConfirm:= bConfirm);
alarms[92](evtEntry:= Tc_Events.AlarmWord6.b12, bEvt:= Alarms_DB.AlarmWord6.AlarmWord.12, bConfirm:= bConfirm);
//alarms[93]
//alarms[94]
//alarms[95]

// Alarm Word 7 - Charger Alarms
Alarms_DB.AlarmWord7.AlarmWord.0 := Trips_DB.Charger[6].OverTemp;
Alarms_DB.AlarmWord7.AlarmWord.1 := Trips_DB.Charger[6].InterlockOpen;
Alarms_DB.AlarmWord7.AlarmWord.2 := Trips_DB.Charger[6].LoadFaulted;
Alarms_DB.AlarmWord7.AlarmWord.3 := Trips_DB.Charger[7].OverTemp;
Alarms_DB.AlarmWord7.AlarmWord.4 := Trips_DB.Charger[7].InterlockOpen;
Alarms_DB.AlarmWord7.AlarmWord.5 := Trips_DB.Charger[7].LoadFaulted;
Alarms_DB.AlarmWord7.AlarmWord.6 := Trips_DB.Charger[8].OverTemp;
Alarms_DB.AlarmWord7.AlarmWord.7 := Trips_DB.Charger[8].InterlockOpen;
Alarms_DB.AlarmWord7.AlarmWord.8 := Trips_DB.Charger[8].LoadFaulted;
Alarms_DB.AlarmWord7.AlarmWord.9 := Trips_DB.AnyChargerOverTemp; 
Alarms_DB.AlarmWord7.AlarmWord.10 := Trips_DB.AnyChargerLoadFault; 
Alarms_DB.AlarmWord7.AlarmWord.11 := Trips_DB.AnySystemTripped; 
Alarms_DB.AlarmWord7.AlarmWord.12 := Trips_DB.MachineGNDrlyFailed; 
Alarms_DB.AlarmWord7.AlarmWord.13 := Trips_DB.AnyChargeRlyFail; 
Alarms_DB.AlarmWord7.AlarmWord.14 := Trips_DB.AnyDumpRlyFail; 
Alarms_DB.AlarmWord7.AlarmWord.15 := Trips_DB.AnyLossInhibitSignal; 

// Alarm Word 7 - Msg
alarms[96](evtEntry:= Tc_Events.AlarmWord7.b0, bEvt:= Alarms_DB.AlarmWord7.AlarmWord.0, bConfirm:= bConfirm);
alarms[97](evtEntry:= Tc_Events.AlarmWord7.b1, bEvt:= Alarms_DB.AlarmWord7.AlarmWord.1, bConfirm:= bConfirm);
alarms[98](evtEntry:= Tc_Events.AlarmWord7.b2, bEvt:= Alarms_DB.AlarmWord7.AlarmWord.2, bConfirm:= bConfirm);
alarms[99](evtEntry:= Tc_Events.AlarmWord7.b3, bEvt:= Alarms_DB.AlarmWord7.AlarmWord.3, bConfirm:= bConfirm);
alarms[100](evtEntry:= Tc_Events.AlarmWord7.b4, bEvt:= Alarms_DB.AlarmWord7.AlarmWord.4, bConfirm:= bConfirm);
alarms[101](evtEntry:= Tc_Events.AlarmWord7.b5, bEvt:= Alarms_DB.AlarmWord7.AlarmWord.5, bConfirm:= bConfirm);
alarms[102](evtEntry:= Tc_Events.AlarmWord7.b6, bEvt:= Alarms_DB.AlarmWord7.AlarmWord.6, bConfirm:= bConfirm);
alarms[103](evtEntry:= Tc_Events.AlarmWord7.b7, bEvt:= Alarms_DB.AlarmWord7.AlarmWord.7, bConfirm:= bConfirm);
alarms[104](evtEntry:= Tc_Events.AlarmWord7.b8, bEvt:= Alarms_DB.AlarmWord7.AlarmWord.8, bConfirm:= bConfirm);
alarms[105](evtEntry:= Tc_Events.AlarmWord7.b9, bEvt:= Alarms_DB.AlarmWord7.AlarmWord.9, bConfirm:= bConfirm);
alarms[106](evtEntry:= Tc_Events.AlarmWord7.b10, bEvt:= Alarms_DB.AlarmWord7.AlarmWord.10, bConfirm:= bConfirm);
alarms[107](evtEntry:= Tc_Events.AlarmWord7.b11, bEvt:= Alarms_DB.AlarmWord7.AlarmWord.11, bConfirm:= bConfirm);
alarms[108](evtEntry:= Tc_Events.AlarmWord7.b12, bEvt:= Alarms_DB.AlarmWord7.AlarmWord.12, bConfirm:= bConfirm);
alarms[109](evtEntry:= Tc_Events.AlarmWord7.b13, bEvt:= Alarms_DB.AlarmWord7.AlarmWord.13, bConfirm:= bConfirm);
alarms[110](evtEntry:= Tc_Events.AlarmWord7.b14, bEvt:= Alarms_DB.AlarmWord7.AlarmWord.14, bConfirm:= bConfirm);
alarms[111] (evtEntry:= Tc_Events.AlarmWord7.b15, bEvt:= Alarms_DB.AlarmWord7.AlarmWord.15, bConfirm:= bConfirm);


//Alarm Word 8 
Alarms_DB.AlarmWord8.AlarmWord.0 := NOT Trips_DB.AllDCpsuOK;
Alarms_DB.AlarmWord8.AlarmWord.1 := Trips_DB.AnyChargerFaulted;
Alarms_DB.AlarmWord8.AlarmWord.2 := Trips_DB.AnyLossHVONsignal;
Alarms_DB.AlarmWord8.AlarmWord.3 := NOT Trips_DB.NoFaultDetected;
Alarms_DB.AlarmWord8.AlarmWord.4 := LCP.Section[1].Peak.ShortContact1unknown;
Alarms_DB.AlarmWord8.AlarmWord.5 := LCP.Section[1].Peak.ShortContact2unknown;
Alarms_DB.AlarmWord8.AlarmWord.6 := LCP.Section[2].Peak.ShortContact1unknown;
Alarms_DB.AlarmWord8.AlarmWord.7 := LCP.Section[2].Peak.ShortContact2unknown;
Alarms_DB.AlarmWord8.AlarmWord.8 := LCP.Section[3].Peak.ShortContact1unknown;
Alarms_DB.AlarmWord8.AlarmWord.9 := LCP.Section[3].Peak.ShortContact2unknown;
Alarms_DB.AlarmWord8.AlarmWord.10 := LCP.Section[1].Sust.ShortContact1unknown;
Alarms_DB.AlarmWord8.AlarmWord.11 := LCP.Section[1].Sust.ShortContact2unknown;
Alarms_DB.AlarmWord8.AlarmWord.12 := LCP.Section[2].Sust.ShortContact1unknown;
Alarms_DB.AlarmWord8.AlarmWord.13 := LCP.Section[2].Sust.ShortContact2unknown;
Alarms_DB.AlarmWord8.AlarmWord.14 := LCP.Section[3].Sust.ShortContact1unknown;
Alarms_DB.AlarmWord8.AlarmWord.15 := LCP.Section[3].Sust.ShortContact2unknown;

//Alarm Word 8 - msg
alarms[112](evtEntry:= Tc_Events.AlarmWord8.b0, bEvt:= Alarms_DB.AlarmWord8.AlarmWord.0, bConfirm:= bConfirm);
alarms[113](evtEntry:= Tc_Events.AlarmWord8.b1, bEvt:= Alarms_DB.AlarmWord8.AlarmWord.1, bConfirm:= bConfirm);
alarms[114](evtEntry:= Tc_Events.AlarmWord8.b2, bEvt:= Alarms_DB.AlarmWord8.AlarmWord.2, bConfirm:= bConfirm);
alarms[115](evtEntry:= Tc_Events.AlarmWord8.b3, bEvt:= Alarms_DB.AlarmWord8.AlarmWord.3, bConfirm:= bConfirm);
alarms[116](evtEntry:= Tc_Events.AlarmWord8.b4, bEvt:= Alarms_DB.AlarmWord8.AlarmWord.4, bConfirm:= bConfirm);
alarms[117](evtEntry:= Tc_Events.AlarmWord8.b5, bEvt:= Alarms_DB.AlarmWord8.AlarmWord.5, bConfirm:= bConfirm);
alarms[118](evtEntry:= Tc_Events.AlarmWord8.b6, bEvt:= Alarms_DB.AlarmWord8.AlarmWord.6, bConfirm:= bConfirm);
alarms[119](evtEntry:= Tc_Events.AlarmWord8.b7, bEvt:= Alarms_DB.AlarmWord8.AlarmWord.7, bConfirm:= bConfirm);
alarms[120](evtEntry:= Tc_Events.AlarmWord8.b8, bEvt:= Alarms_DB.AlarmWord8.AlarmWord.8, bConfirm:= bConfirm);
alarms[121](evtEntry:= Tc_Events.AlarmWord8.b9, bEvt:= Alarms_DB.AlarmWord8.AlarmWord.9, bConfirm:= bConfirm);
alarms[122](evtEntry:= Tc_Events.AlarmWord8.b10, bEvt:= Alarms_DB.AlarmWord8.AlarmWord.10, bConfirm:= bConfirm);
alarms[123](evtEntry:= Tc_Events.AlarmWord8.b11, bEvt:= Alarms_DB.AlarmWord8.AlarmWord.11, bConfirm:= bConfirm);
alarms[124](evtEntry:= Tc_Events.AlarmWord8.b12, bEvt:= Alarms_DB.AlarmWord8.AlarmWord.12, bConfirm:= bConfirm);
alarms[125](evtEntry:= Tc_Events.AlarmWord8.b13, bEvt:= Alarms_DB.AlarmWord8.AlarmWord.13, bConfirm:= bConfirm);
alarms[126](evtEntry:= Tc_Events.AlarmWord8.b14, bEvt:= Alarms_DB.AlarmWord8.AlarmWord.14, bConfirm:= bConfirm);
alarms[127] (evtEntry:= Tc_Events.AlarmWord8.b15, bEvt:= Alarms_DB.AlarmWord8.AlarmWord.15, bConfirm:= bConfirm);

//Alarm Word 9 
Alarms_DB.AlarmWord9.AlarmWord.0 := LCP.Section[4].Form.ShortContact1unknown;
Alarms_DB.AlarmWord9.AlarmWord.1 := LCP.Section[4].Form.ShortContact2unknown;
Alarms_DB.AlarmWord9.AlarmWord.2 := LCP.Section[4].Form.FormTrigShortContactUnknown;
Alarms_DB.AlarmWord9.AlarmWord.3 := LCP.Section[4].Form.PreFormTrigShortContactUnknown;
Alarms_DB.AlarmWord9.AlarmWord.4 := NOT Permissives_DB.NoShortingUnknowns;
Alarms_DB.AlarmWord9.AlarmWord.5 := NOT Permissives_DB.NoInterlockPressureLoss;
Alarms_DB.AlarmWord9.AlarmWord.6 := NOT Permissives_DB.SafetyOK;
//Alarms_DB.AlarmWord9.AlarmWord.7 := 
//Alarms_DB.AlarmWord9.AlarmWord.8 := 
//Alarms_DB.AlarmWord9.AlarmWord.9 := 
//Alarms_DB.AlarmWord9.AlarmWord.10 := 
//Alarms_DB.AlarmWord9.AlarmWord.11 := 
//Alarms_DB.AlarmWord9.AlarmWord.12 := 
//Alarms_DB.AlarmWord9.AlarmWord.13 := 
//Alarms_DB.AlarmWord9.AlarmWord.14 := 
Alarms_DB.AlarmWord9.AlarmWord.15 := Trips_DB.DumpTimerRunout;

//Alarm Word 9 - msg
alarms[112](evtEntry:= Tc_Events.AlarmWord9.b0, bEvt:= Alarms_DB.AlarmWord9.AlarmWord.0, bConfirm:= bConfirm);
alarms[113](evtEntry:= Tc_Events.AlarmWord9.b1, bEvt:= Alarms_DB.AlarmWord9.AlarmWord.1, bConfirm:= bConfirm);
alarms[114](evtEntry:= Tc_Events.AlarmWord9.b2, bEvt:= Alarms_DB.AlarmWord9.AlarmWord.2, bConfirm:= bConfirm);
alarms[115](evtEntry:= Tc_Events.AlarmWord9.b3, bEvt:= Alarms_DB.AlarmWord9.AlarmWord.3, bConfirm:= bConfirm);
alarms[116](evtEntry:= Tc_Events.AlarmWord9.b4, bEvt:= Alarms_DB.AlarmWord9.AlarmWord.4, bConfirm:= bConfirm);
alarms[117](evtEntry:= Tc_Events.AlarmWord9.b5, bEvt:= Alarms_DB.AlarmWord9.AlarmWord.5, bConfirm:= bConfirm);
alarms[118](evtEntry:= Tc_Events.AlarmWord9.b6, bEvt:= Alarms_DB.AlarmWord9.AlarmWord.6, bConfirm:= bConfirm);
//alarms[119](evtEntry:= Tc_Events.AlarmWord9.b7, bEvt:= Alarms_DB.AlarmWord9.AlarmWord.7, bConfirm:= bConfirm);
//alarms[120](evtEntry:= Tc_Events.AlarmWord9.b8, bEvt:= Alarms_DB.AlarmWord9.AlarmWord.8, bConfirm:= bConfirm);
//alarms[121](evtEntry:= Tc_Events.AlarmWord9.b9, bEvt:= Alarms_DB.AlarmWord9.AlarmWord.9, bConfirm:= bConfirm);
//alarms[122](evtEntry:= Tc_Events.AlarmWord9.b10, bEvt:= Alarms_DB.AlarmWord9.AlarmWord.10, bConfirm:= bConfirm);
//alarms[123](evtEntry:= Tc_Events.AlarmWord9.b11, bEvt:= Alarms_DB.AlarmWord9.AlarmWord.11, bConfirm:= bConfirm);
//alarms[124](evtEntry:= Tc_Events.AlarmWord9.b12, bEvt:= Alarms_DB.AlarmWord9.AlarmWord.12, bConfirm:= bConfirm);
//alarms[125](evtEntry:= Tc_Events.AlarmWord9.b13, bEvt:= Alarms_DB.AlarmWord9.AlarmWord.13, bConfirm:= bConfirm);
//alarms[126](evtEntry:= Tc_Events.AlarmWord9.b14, bEvt:= Alarms_DB.AlarmWord9.AlarmWord.14, bConfirm:= bConfirm);
alarms[127] (evtEntry:= Tc_Events.AlarmWord9.b15, bEvt:= Alarms_DB.AlarmWord9.AlarmWord.15, bConfirm:= bConfirm);

//Alarm Word 11
(* uncomment this when instrument is ready
Alarms_DB.AlarmWord_11.AlarmWord.0 := Devices.Coil1.AC_Interlock_RlyOpen;
Alarms_DB.AlarmWord_11.AlarmWord.1 := Devices.Coil2.AC_Interlock_RlyOpen;
Alarms_DB.AlarmWord_11.AlarmWord.2 := Devices.Coil3.AC_Interlock_RlyOpen;
Alarms_DB.AlarmWord_11.AlarmWord.3 := Devices.Coil4.AC_Interlock_RlyOpen;
Alarms_DB.AlarmWord_11.AlarmWord.4 := Devices.Coil5.AC_Interlock_RlyOpen;
Alarms_DB.AlarmWord_11.AlarmWord.5 := Devices.Coil6.AC_Interlock_RlyOpen;
Alarms_DB.AlarmWord_11.AlarmWord.6 := Devices.Coil7.AC_Interlock_RlyOpen;
Alarms_DB.AlarmWord_11.AlarmWord.7 := Devices.Coil8.AC_Interlock_RlyOpen;
Alarms_DB.AlarmWord_11.AlarmWord.8 := Devices.Coil9.AC_Interlock_RlyOpen;
Alarms_DB.AlarmWord_11.AlarmWord.9 := Devices.Coil10.AC_Interlock_RlyOpen;
Alarms_DB.AlarmWord_11.AlarmWord.10 := NOT Permissives.AllInterlock_Closed;
*)
//Alarm Word 11 - msg
(*alarms[160](evtEntry:= Tc_Events.AlarmWord11.b0, bEvt:= Alarms_DB.AlarmWord_11.AlarmWord.0, bConfirm:= bConfirm);
alarms[161](evtEntry:= Tc_Events.AlarmWord11.b1, bEvt:= Alarms_DB.AlarmWord_11.AlarmWord.1, bConfirm:= bConfirm);
alarms[162](evtEntry:= Tc_Events.AlarmWord11.b2, bEvt:= Alarms_DB.AlarmWord_11.AlarmWord.2, bConfirm:= bConfirm);
alarms[163](evtEntry:= Tc_Events.AlarmWord11.b3, bEvt:= Alarms_DB.AlarmWord_11.AlarmWord.3, bConfirm:= bConfirm);
alarms[164](evtEntry:= Tc_Events.AlarmWord11.b4, bEvt:= Alarms_DB.AlarmWord_11.AlarmWord.4, bConfirm:= bConfirm);
alarms[165](evtEntry:= Tc_Events.AlarmWord11.b5, bEvt:= Alarms_DB.AlarmWord_11.AlarmWord.5, bConfirm:= bConfirm);
alarms[166](evtEntry:= Tc_Events.AlarmWord11.b6, bEvt:= Alarms_DB.AlarmWord_11.AlarmWord.6, bConfirm:= bConfirm);
alarms[167](evtEntry:= Tc_Events.AlarmWord11.b7, bEvt:= Alarms_DB.AlarmWord_11.AlarmWord.7, bConfirm:= bConfirm);
alarms[168](evtEntry:= Tc_Events.AlarmWord11.b8, bEvt:= Alarms_DB.AlarmWord_11.AlarmWord.8, bConfirm:= bConfirm);
alarms[169](evtEntry:= Tc_Events.AlarmWord11.b9, bEvt:= Alarms_DB.AlarmWord_11.AlarmWord.9, bConfirm:= bConfirm);
alarms[170](evtEntry:= Tc_Events.AlarmWord11.b10, bEvt:= Alarms_DB.AlarmWord_11.AlarmWord.10, bConfirm:= bConfirm);

//Alarm Word 12




//Alarm Word 22
//uncomment this when instrument is ready - commented out for testing only
Alarms_DB.AlarmWord_22.AlarmWord.0 := MCP_IO.MasterStopPB_Pressed; //NC
(*//Alarms_DB1.AlarmWord_22.AlarmWord.1 := Devices.Coil[1].Local_EstopPB_Pressed; //NC
Alarms_DB1.AlarmWord_22.AlarmWord.2 := Devices.Coil2.Local_EstopPB_Pressed; //NC
Alarms_DB1.AlarmWord_22.AlarmWord.3 := Devices.Coil3.Local_EstopPB_Pressed; //NC
Alarms_DB1.AlarmWord_22.AlarmWord.4 := Devices.Coil4.Local_EstopPB_Pressed; //NC
Alarms_DB1.AlarmWord_22.AlarmWord.5 := Devices.Coil5.Local_EstopPB_Pressed; //NC
Alarms_DB1.AlarmWord_22.AlarmWord.6 := Devices.Coil6.Local_EstopPB_Pressed; //NC
Alarms_DB1.AlarmWord_22.AlarmWord.7 := Devices.Coil7.Local_EstopPB_Pressed; //NC
Alarms_DB1.AlarmWord_22.AlarmWord.8 := Devices.Coil8.Local_EstopPB_Pressed; //NC
Alarms_DB1.AlarmWord_22.AlarmWord.9 := Devices.Coil9.Local_EstopPB_Pressed; //NC
Alarms_DB1.AlarmWord_22.AlarmWord.10 := Devices.Coil10.Local_EstopPB_Pressed; //NC
//Alarms_DB1.AlarmWord_22.AlarmWord.11 := NOT Input.R1_01_02; //0 = Manual Mode , 1 = Auto mode
//Alarms_DB1.AlarmWord_22.AlarmWord.12 := NOT Input.R1_01_01; //0 = circuit broken , 1 = circuit ok
//Alarms_DB1.AlarmWord_22.AlarmWord.13 := Spare
//Alarms_DB1.AlarmWord_22.AlarmWord.14 := Spare
//Alarms_DB1.AlarmWord_22.AlarmWord.15 := Spare
*)

//Alarm Word 22 msg
alarms[336](evtEntry:= Tc_Events.AlarmWord22.b0, bEvt:= Alarms_DB.AlarmWord_22.AlarmWord.0, bConfirm:= bConfirm);
alarms[337](evtEntry:= Tc_Events.AlarmWord22.b1, bEvt:= Alarms_DB.AlarmWord_22.AlarmWord.1, bConfirm:= bConfirm);
alarms[338](evtEntry:= Tc_Events.AlarmWord22.b2, bEvt:= Alarms_DB.AlarmWord_22.AlarmWord.2, bConfirm:= bConfirm);
alarms[339](evtEntry:= Tc_Events.AlarmWord22.b3, bEvt:= Alarms_DB.AlarmWord_22.AlarmWord.3, bConfirm:= bConfirm);
alarms[340](evtEntry:= Tc_Events.AlarmWord22.b4, bEvt:= Alarms_DB.AlarmWord_22.AlarmWord.4, bConfirm:= bConfirm);
alarms[341](evtEntry:= Tc_Events.AlarmWord22.b5, bEvt:= Alarms_DB.AlarmWord_22.AlarmWord.5, bConfirm:= bConfirm);
alarms[342](evtEntry:= Tc_Events.AlarmWord22.b6, bEvt:= Alarms_DB.AlarmWord_22.AlarmWord.6, bConfirm:= bConfirm);
alarms[343](evtEntry:= Tc_Events.AlarmWord22.b7, bEvt:= Alarms_DB.AlarmWord_22.AlarmWord.7, bConfirm:= bConfirm);
alarms[344](evtEntry:= Tc_Events.AlarmWord22.b8, bEvt:= Alarms_DB.AlarmWord_22.AlarmWord.8, bConfirm:= bConfirm);
alarms[345](evtEntry:= Tc_Events.AlarmWord22.b9, bEvt:= Alarms_DB.AlarmWord_22.AlarmWord.9, bConfirm:= bConfirm);
alarms[346](evtEntry:= Tc_Events.AlarmWord22.b10, bEvt:= Alarms_DB.AlarmWord_22.AlarmWord.10, bConfirm:= bConfirm);
alarms[347](evtEntry:= Tc_Events.AlarmWord22.b11, bEvt:= Alarms_DB.AlarmWord_22.AlarmWord.11, bConfirm:= bConfirm);
alarms[348](evtEntry:= Tc_Events.AlarmWord22.b12, bEvt:= Alarms_DB.AlarmWord_22.AlarmWord.12, bConfirm:= bConfirm);

//Alarm Word 23
(* uncomment when instrument is ready
Alarms_DB.AlarmWord_23.AlarmWord.0 := Trips_DB.Coil[1].ChargeRelay_FailtoClose; 
Alarms_DB.AlarmWord_23.AlarmWord.1 := Trips_DB.Coil[1].ChargeRelay_FailtoOpen;
Alarms_DB.AlarmWord_23.AlarmWord.2 := Trips_DB.Coil[2].ChargeRelay_FailtoClose;
Alarms_DB.AlarmWord_23.AlarmWord.3 := Trips_DB.Coil[2].ChargeRelay_FailtoOpen;
Alarms_DB.AlarmWord_23.AlarmWord.4 := Trips_DB.Coil[3].ChargeRelay_FailtoClose;
Alarms_DB.AlarmWord_23.AlarmWord.5 := Trips_DB.Coil[3].ChargeRelay_FailtoOpen;
Alarms_DB.AlarmWord_23.AlarmWord.6 := Trips_DB.Coil[4].ChargeRelay_FailtoClose;
Alarms_DB.AlarmWord_23.AlarmWord.7 := Trips_DB.Coil[4].ChargeRelay_FailtoOpen;
Alarms_DB.AlarmWord_23.AlarmWord.8 := Trips_DB.Coil[5].ChargeRelay_FailtoClose;
Alarms_DB.AlarmWord_23.AlarmWord.9 := Trips_DB.Coil[5].ChargeRelay_FailtoOpen;
Alarms_DB.AlarmWord_23.AlarmWord.10 := Trips_DB.Coil[6].ChargeRelay_FailtoClose;
Alarms_DB.AlarmWord_23.AlarmWord.11 := Trips_DB.Coil[6].ChargeRelay_FailtoOpen;
Alarms_DB.AlarmWord_23.AlarmWord.12 := Trips_DB.Coil[7].ChargeRelay_FailtoClose;
Alarms_DB.AlarmWord_23.AlarmWord.13 := Trips_DB.Coil[7].ChargeRelay_FailtoOpen;
Alarms_DB.AlarmWord_23.AlarmWord.14 := Trips_DB.Coil[8].ChargeRelay_FailtoClose;
Alarms_DB.AlarmWord_23.AlarmWord.15 := Trips_DB.Coil[9].ChargeRelay_FailtoOpen;
*)
//Alarm Word 23 msg
alarms[352](evtEntry:= Tc_Events.AlarmWord23.b0, bEvt:= Alarms_DB.AlarmWord_23.AlarmWord.0, bConfirm:= bConfirm);
alarms[353](evtEntry:= Tc_Events.AlarmWord23.b1, bEvt:= Alarms_DB.AlarmWord_23.AlarmWord.1, bConfirm:= bConfirm);
alarms[354](evtEntry:= Tc_Events.AlarmWord23.b2, bEvt:= Alarms_DB.AlarmWord_23.AlarmWord.2, bConfirm:= bConfirm);
alarms[355](evtEntry:= Tc_Events.AlarmWord23.b3, bEvt:= Alarms_DB.AlarmWord_23.AlarmWord.3, bConfirm:= bConfirm);
alarms[356](evtEntry:= Tc_Events.AlarmWord23.b4, bEvt:= Alarms_DB.AlarmWord_23.AlarmWord.4, bConfirm:= bConfirm);
alarms[357](evtEntry:= Tc_Events.AlarmWord23.b5, bEvt:= Alarms_DB.AlarmWord_23.AlarmWord.5, bConfirm:= bConfirm);
alarms[358](evtEntry:= Tc_Events.AlarmWord23.b6, bEvt:= Alarms_DB.AlarmWord_23.AlarmWord.6, bConfirm:= bConfirm);
alarms[359](evtEntry:= Tc_Events.AlarmWord23.b7, bEvt:= Alarms_DB.AlarmWord_23.AlarmWord.7, bConfirm:= bConfirm);
alarms[360](evtEntry:= Tc_Events.AlarmWord23.b8, bEvt:= Alarms_DB.AlarmWord_23.AlarmWord.8, bConfirm:= bConfirm);
alarms[361](evtEntry:= Tc_Events.AlarmWord23.b9, bEvt:= Alarms_DB.AlarmWord_23.AlarmWord.9, bConfirm:= bConfirm);
alarms[362](evtEntry:= Tc_Events.AlarmWord23.b10, bEvt:= Alarms_DB.AlarmWord_23.AlarmWord.10, bConfirm:= bConfirm);
alarms[363](evtEntry:= Tc_Events.AlarmWord23.b11, bEvt:= Alarms_DB.AlarmWord_23.AlarmWord.11, bConfirm:= bConfirm);
alarms[364](evtEntry:= Tc_Events.AlarmWord23.b12, bEvt:= Alarms_DB.AlarmWord_23.AlarmWord.12, bConfirm:= bConfirm);
alarms[365](evtEntry:= Tc_Events.AlarmWord23.b13, bEvt:= Alarms_DB.AlarmWord_23.AlarmWord.13, bConfirm:= bConfirm);
alarms[366](evtEntry:= Tc_Events.AlarmWord23.b14, bEvt:= Alarms_DB.AlarmWord_23.AlarmWord.14, bConfirm:= bConfirm);
alarms[367](evtEntry:= Tc_Events.AlarmWord23.b15, bEvt:= Alarms_DB.AlarmWord_23.AlarmWord.15, bConfirm:= bConfirm);

//Alarm Word 24
(* uncomment when instrument is ready
Alarms_DB.AlarmWord_24.AlarmWord.0 := Trips_DB.Coil[9].ChargeRelay_FailtoClose; 
Alarms_DB.AlarmWord_24.AlarmWord.1 := Trips_DB.Coil[9].ChargeRelay_FailtoOpen;
Alarms_DB.AlarmWord_24.AlarmWord.2 := Trips_DB.Coil[10].ChargeRelay_FailtoClose;
Alarms_DB.AlarmWord_24.AlarmWord.3 := Trips_DB.Coil[10].ChargeRelay_FailtoOpen;
Alarms_DB.AlarmWord_24.AlarmWord.4 := Trips_DB.Coil[1].ACInterlockRelayFailedtoClose;
Alarms_DB.AlarmWord_24.AlarmWord.5 := Trips_DB.Coil[1].ACInterlockRelayFailedtoOpen;
Alarms_DB.AlarmWord_24.AlarmWord.6 := Trips_DB.Coil[2].ACInterlockRelayFailedtoClose;
Alarms_DB.AlarmWord_24.AlarmWord.7 := Trips_DB.Coil[2].ACInterlockRelayFailedtoOpen;
Alarms_DB.AlarmWord_24.AlarmWord.8 := Trips_DB.Coil[3].ACInterlockRelayFailedtoClose;
Alarms_DB.AlarmWord_24.AlarmWord.9 := Trips_DB.Coil[3].ACInterlockRelayFailedtoOpen;
Alarms_DB.AlarmWord_24.AlarmWord.10 := Trips_DB.Coil[4].ACInterlockRelayFailedtoClose;
Alarms_DB.AlarmWord_24.AlarmWord.11 := Trips_DB.Coil[4].ACInterlockRelayFailedtoOpen;
Alarms_DB.AlarmWord_24.AlarmWord.12 := Trips_DB.Coil[5].ACInterlockRelayFailedtoClose;
Alarms_DB.AlarmWord_24.AlarmWord.13 := Trips_DB.Coil[5].ACInterlockRelayFailedtoOpen;
Alarms_DB.AlarmWord_24.AlarmWord.14 := Trips_DB.Coil[6].ACInterlockRelayFailedtoClose;
Alarms_DB.AlarmWord_24.AlarmWord.15 := Trips_DB.Coil[6].ACInterlockRelayFailedtoOpen;
*)
//Alarm Word 24 msg
alarms[368](evtEntry:= Tc_Events.AlarmWord24.b0, bEvt:= Alarms_DB.AlarmWord_24.AlarmWord.0, bConfirm:= bConfirm);
alarms[369](evtEntry:= Tc_Events.AlarmWord24.b1, bEvt:= Alarms_DB.AlarmWord_24.AlarmWord.1, bConfirm:= bConfirm);
alarms[370](evtEntry:= Tc_Events.AlarmWord24.b2, bEvt:= Alarms_DB.AlarmWord_24.AlarmWord.2, bConfirm:= bConfirm);
alarms[371](evtEntry:= Tc_Events.AlarmWord24.b3, bEvt:= Alarms_DB.AlarmWord_24.AlarmWord.3, bConfirm:= bConfirm);
alarms[372](evtEntry:= Tc_Events.AlarmWord24.b4, bEvt:= Alarms_DB.AlarmWord_24.AlarmWord.4, bConfirm:= bConfirm);
alarms[373](evtEntry:= Tc_Events.AlarmWord24.b5, bEvt:= Alarms_DB.AlarmWord_24.AlarmWord.5, bConfirm:= bConfirm);
alarms[374](evtEntry:= Tc_Events.AlarmWord24.b6, bEvt:= Alarms_DB.AlarmWord_24.AlarmWord.6, bConfirm:= bConfirm);
alarms[375](evtEntry:= Tc_Events.AlarmWord24.b7, bEvt:= Alarms_DB.AlarmWord_24.AlarmWord.7, bConfirm:= bConfirm);
alarms[376](evtEntry:= Tc_Events.AlarmWord24.b8, bEvt:= Alarms_DB.AlarmWord_24.AlarmWord.8, bConfirm:= bConfirm);
alarms[377](evtEntry:= Tc_Events.AlarmWord24.b9, bEvt:= Alarms_DB.AlarmWord_24.AlarmWord.9, bConfirm:= bConfirm);
alarms[378](evtEntry:= Tc_Events.AlarmWord24.b10, bEvt:= Alarms_DB.AlarmWord_24.AlarmWord.10, bConfirm:= bConfirm);
alarms[379](evtEntry:= Tc_Events.AlarmWord24.b11, bEvt:= Alarms_DB.AlarmWord_24.AlarmWord.11, bConfirm:= bConfirm);
alarms[380](evtEntry:= Tc_Events.AlarmWord24.b12, bEvt:= Alarms_DB.AlarmWord_24.AlarmWord.12, bConfirm:= bConfirm);
alarms[381](evtEntry:= Tc_Events.AlarmWord24.b13, bEvt:= Alarms_DB.AlarmWord_24.AlarmWord.13, bConfirm:= bConfirm);
alarms[382](evtEntry:= Tc_Events.AlarmWord24.b14, bEvt:= Alarms_DB.AlarmWord_24.AlarmWord.14, bConfirm:= bConfirm);
alarms[383](evtEntry:= Tc_Events.AlarmWord24.b15, bEvt:= Alarms_DB.AlarmWord_24.AlarmWord.15, bConfirm:= bConfirm);

//Alarm Word 25
(* uncomment when instrument is ready
Alarms_DB.AlarmWord_25.AlarmWord.0 := Trips_DB.Coil[7].ACInterlockRelayFailedtoClose;
Alarms_DB.AlarmWord_25.AlarmWord.1 := Trips_DB.Coil[7].ACInterlockRelayFailedtoOpen;
Alarms_DB.AlarmWord_25.AlarmWord.2 := Trips_DB.Coil[8].ACInterlockRelayFailedtoClose;
Alarms_DB.AlarmWord_25.AlarmWord.3 := Trips_DB.Coil[8].ACInterlockRelayFailedtoOpen;
Alarms_DB.AlarmWord_25.AlarmWord.4 := Trips_DB.Coil[9].ACInterlockRelayFailedtoClose;
Alarms_DB.AlarmWord_25.AlarmWord.5 := Trips_DB.Coil[9].ACInterlockRelayFailedtoOpen;
Alarms_DB.AlarmWord_25.AlarmWord.6 := Trips_DB.Coil[10].ACInterlockRelayFailedtoClose;
Alarms_DB.AlarmWord_25.AlarmWord.7 := Trips_DB.Coil[10].ACInterlockRelayFailedtoOpen;
Alarms_DB.AlarmWord_25.AlarmWord.8 := Trips_DB.Coil[1].DumpRelay1_FailtoClose;
Alarms_DB.AlarmWord_25.AlarmWord.9 := Trips_DB.Coil[1].DumpRelay1_FailtoOpen;
Alarms_DB.AlarmWord_25.AlarmWord.10 := Trips_DB.Coil[2].DumpRelay1_FailtoClose;
Alarms_DB.AlarmWord_25.AlarmWord.11 := Trips_DB.Coil[2].DumpRelay1_FailtoOpen;
Alarms_DB.AlarmWord_25.AlarmWord.12 := Trips_DB.Coil[3].DumpRelay1_FailtoClose;
Alarms_DB.AlarmWord_25.AlarmWord.13 := Trips_DB.Coil[3].DumpRelay1_FailtoOpen;
Alarms_DB.AlarmWord_25.AlarmWord.14 := Trips_DB.Coil[4].DumpRelay1_FailtoClose;
Alarms_DB.AlarmWord_25.AlarmWord.15 := Trips_DB.Coil[4].DumpRelay1_FailtoOpen;
*)
//Alarm Word 25 msg
alarms[384](evtEntry:= Tc_Events.AlarmWord25.b0, bEvt:= Alarms_DB.AlarmWord_25.AlarmWord.0, bConfirm:= bConfirm);
alarms[385](evtEntry:= Tc_Events.AlarmWord25.b1, bEvt:= Alarms_DB.AlarmWord_25.AlarmWord.1, bConfirm:= bConfirm);
alarms[386](evtEntry:= Tc_Events.AlarmWord25.b2, bEvt:= Alarms_DB.AlarmWord_25.AlarmWord.2, bConfirm:= bConfirm);
alarms[387](evtEntry:= Tc_Events.AlarmWord25.b3, bEvt:= Alarms_DB.AlarmWord_25.AlarmWord.3, bConfirm:= bConfirm);
alarms[388](evtEntry:= Tc_Events.AlarmWord25.b4, bEvt:= Alarms_DB.AlarmWord_25.AlarmWord.4, bConfirm:= bConfirm);
alarms[389](evtEntry:= Tc_Events.AlarmWord25.b5, bEvt:= Alarms_DB.AlarmWord_25.AlarmWord.5, bConfirm:= bConfirm);
alarms[390](evtEntry:= Tc_Events.AlarmWord25.b6, bEvt:= Alarms_DB.AlarmWord_25.AlarmWord.6, bConfirm:= bConfirm);
alarms[391](evtEntry:= Tc_Events.AlarmWord25.b7, bEvt:= Alarms_DB.AlarmWord_25.AlarmWord.7, bConfirm:= bConfirm);
alarms[392](evtEntry:= Tc_Events.AlarmWord25.b8, bEvt:= Alarms_DB.AlarmWord_25.AlarmWord.8, bConfirm:= bConfirm);
alarms[393](evtEntry:= Tc_Events.AlarmWord25.b9, bEvt:= Alarms_DB.AlarmWord_25.AlarmWord.9, bConfirm:= bConfirm);
alarms[394](evtEntry:= Tc_Events.AlarmWord25.b10, bEvt:= Alarms_DB.AlarmWord_25.AlarmWord.10, bConfirm:= bConfirm);
alarms[395](evtEntry:= Tc_Events.AlarmWord25.b11, bEvt:= Alarms_DB.AlarmWord_25.AlarmWord.11, bConfirm:= bConfirm);
alarms[396](evtEntry:= Tc_Events.AlarmWord25.b12, bEvt:= Alarms_DB.AlarmWord_25.AlarmWord.12, bConfirm:= bConfirm);
alarms[397](evtEntry:= Tc_Events.AlarmWord25.b13, bEvt:= Alarms_DB.AlarmWord_25.AlarmWord.13, bConfirm:= bConfirm);
alarms[398](evtEntry:= Tc_Events.AlarmWord25.b14, bEvt:= Alarms_DB.AlarmWord_25.AlarmWord.14, bConfirm:= bConfirm);
alarms[399](evtEntry:= Tc_Events.AlarmWord25.b15, bEvt:= Alarms_DB.AlarmWord_25.AlarmWord.15, bConfirm:= bConfirm);

//Alarm Word 26
(* uncomment when instrument is ready
Alarms_DB.AlarmWord_26.AlarmWord.0 := Trips_DB.Coil[5].DumpRelay1_FailtoClose;
Alarms_DB.AlarmWord_26.AlarmWord.1 := Trips_DB.Coil[5].DumpRelay1_FailtoOpen;
Alarms_DB.AlarmWord_26.AlarmWord.2 := Trips_DB.Coil[6].DumpRelay1_FailtoClose;
Alarms_DB.AlarmWord_26.AlarmWord.3 := Trips_DB.Coil[6].DumpRelay1_FailtoOpen;
Alarms_DB.AlarmWord_26.AlarmWord.4 := Trips_DB.Coil[7].DumpRelay1_FailtoClose;
Alarms_DB.AlarmWord_26.AlarmWord.5 := Trips_DB.Coil[7].DumpRelay1_FailtoOpen;
Alarms_DB.AlarmWord_26.AlarmWord.6 := Trips_DB.Coil[8].DumpRelay1_FailtoClose;
Alarms_DB.AlarmWord_26.AlarmWord.7 := Trips_DB.Coil[8].DumpRelay1_FailtoOpen;
Alarms_DB.AlarmWord_26.AlarmWord.8 := Trips_DB.Coil[9].DumpRelay1_FailtoClose;
Alarms_DB.AlarmWord_26.AlarmWord.9 := Trips_DB.Coil[9].DumpRelay1_FailtoOpen;
Alarms_DB.AlarmWord_26.AlarmWord.10 := Trips_DB.Coil[10].DumpRelay1_FailtoClose;
Alarms_DB.AlarmWord_26.AlarmWord.11 := Trips_DB.Coil[10].DumpRelay1_FailtoOpen;
Alarms_DB.AlarmWord_26.AlarmWord.12 := Trips_DB.Coil[1].DumpRelay2_FailtoClose;
Alarms_DB.AlarmWord_26.AlarmWord.13 := Trips_DB.Coil[1].DumpRelay2_FailtoOpen;
Alarms_DB.AlarmWord_26.AlarmWord.14 := Trips_DB.Coil[2].DumpRelay2_FailtoClose;
Alarms_DB.AlarmWord_26.AlarmWord.15 := Trips_DB.Coil[2].DumpRelay2_FailtoOpen;
*)
//Alarm Word 26 msg
alarms[400](evtEntry:= Tc_Events.AlarmWord26.b0, bEvt:= Alarms_DB.AlarmWord_26.AlarmWord.0, bConfirm:= bConfirm);
alarms[401](evtEntry:= Tc_Events.AlarmWord26.b1, bEvt:= Alarms_DB.AlarmWord_26.AlarmWord.1, bConfirm:= bConfirm);
alarms[402](evtEntry:= Tc_Events.AlarmWord26.b2, bEvt:= Alarms_DB.AlarmWord_26.AlarmWord.2, bConfirm:= bConfirm);
alarms[403](evtEntry:= Tc_Events.AlarmWord26.b3, bEvt:= Alarms_DB.AlarmWord_26.AlarmWord.3, bConfirm:= bConfirm);
alarms[404](evtEntry:= Tc_Events.AlarmWord26.b4, bEvt:= Alarms_DB.AlarmWord_26.AlarmWord.4, bConfirm:= bConfirm);
alarms[405](evtEntry:= Tc_Events.AlarmWord26.b5, bEvt:= Alarms_DB.AlarmWord_26.AlarmWord.5, bConfirm:= bConfirm);
alarms[406](evtEntry:= Tc_Events.AlarmWord26.b6, bEvt:= Alarms_DB.AlarmWord_26.AlarmWord.6, bConfirm:= bConfirm);
alarms[407](evtEntry:= Tc_Events.AlarmWord26.b7, bEvt:= Alarms_DB.AlarmWord_26.AlarmWord.7, bConfirm:= bConfirm);
alarms[408](evtEntry:= Tc_Events.AlarmWord26.b8, bEvt:= Alarms_DB.AlarmWord_26.AlarmWord.8, bConfirm:= bConfirm);
alarms[409](evtEntry:= Tc_Events.AlarmWord26.b9, bEvt:= Alarms_DB.AlarmWord_26.AlarmWord.9, bConfirm:= bConfirm);
alarms[410](evtEntry:= Tc_Events.AlarmWord26.b10, bEvt:= Alarms_DB.AlarmWord_26.AlarmWord.10, bConfirm:= bConfirm);
alarms[411](evtEntry:= Tc_Events.AlarmWord26.b11, bEvt:= Alarms_DB.AlarmWord_26.AlarmWord.11, bConfirm:= bConfirm);
alarms[412](evtEntry:= Tc_Events.AlarmWord26.b12, bEvt:= Alarms_DB.AlarmWord_26.AlarmWord.12, bConfirm:= bConfirm);
alarms[413](evtEntry:= Tc_Events.AlarmWord26.b13, bEvt:= Alarms_DB.AlarmWord_26.AlarmWord.13, bConfirm:= bConfirm);
alarms[414](evtEntry:= Tc_Events.AlarmWord26.b14, bEvt:= Alarms_DB.AlarmWord_26.AlarmWord.14, bConfirm:= bConfirm);
alarms[415](evtEntry:= Tc_Events.AlarmWord26.b15, bEvt:= Alarms_DB.AlarmWord_26.AlarmWord.15, bConfirm:= bConfirm);

//Alarm Word 27
(* uncomment when instrument is ready
Alarms_DB.AlarmWord_27.AlarmWord.0 := Trips_DB.Coil[3].DumpRelay2_FailtoClose;
Alarms_DB.AlarmWord_27.AlarmWord.1 := Trips_DB.Coil[3].DumpRelay2_FailtoOpen;
Alarms_DB.AlarmWord_27.AlarmWord.2 := Trips_DB.Coil[4].DumpRelay2_FailtoClose;
Alarms_DB.AlarmWord_27.AlarmWord.3 := Trips_DB.Coil[4].DumpRelay2_FailtoOpen;
Alarms_DB.AlarmWord_27.AlarmWord.4 := Trips_DB.Coil[5].DumpRelay2_FailtoClose;
Alarms_DB.AlarmWord_27.AlarmWord.5 := Trips_DB.Coil[5].DumpRelay2_FailtoOpen;
Alarms_DB.AlarmWord_27.AlarmWord.6 := Trips_DB.Coil[6].DumpRelay2_FailtoClose;
Alarms_DB.AlarmWord_27.AlarmWord.7 := Trips_DB.Coil[6].DumpRelay2_FailtoOpen;
Alarms_DB.AlarmWord_27.AlarmWord.8 := Trips_DB.Coil[7].DumpRelay2_FailtoClose;
Alarms_DB.AlarmWord_27.AlarmWord.9 := Trips_DB.Coil[7].DumpRelay2_FailtoOpen;
Alarms_DB.AlarmWord_27.AlarmWord.10 := Trips_DB.Coil[8].DumpRelay2_FailtoClose;
Alarms_DB.AlarmWord_27.AlarmWord.11 := Trips_DB.Coil[8].DumpRelay2_FailtoOpen;
Alarms_DB.AlarmWord_27.AlarmWord.12:= Trips_DB.Coil[9].DumpRelay2_FailtoClose;
Alarms_DB.AlarmWord_27.AlarmWord.13 := Trips_DB.Coil[9].DumpRelay2_FailtoOpen;
Alarms_DB.AlarmWord_27.AlarmWord.14 := Trips_DB.Coil[10].DumpRelay2_FailtoClose;
Alarms_DB.AlarmWord_27.AlarmWord.15 := Trips_DB.Coil[10].DumpRelay2_FailtoOpen;
*)
//Alarm Word 27 msg
alarms[416](evtEntry:= Tc_Events.AlarmWord27.b0, bEvt:= Alarms_DB.AlarmWord_27.AlarmWord.0, bConfirm:= bConfirm);
alarms[417](evtEntry:= Tc_Events.AlarmWord27.b1, bEvt:= Alarms_DB.AlarmWord_27.AlarmWord.1, bConfirm:= bConfirm);
alarms[418](evtEntry:= Tc_Events.AlarmWord27.b2, bEvt:= Alarms_DB.AlarmWord_27.AlarmWord.2, bConfirm:= bConfirm);
alarms[419](evtEntry:= Tc_Events.AlarmWord27.b3, bEvt:= Alarms_DB.AlarmWord_27.AlarmWord.3, bConfirm:= bConfirm);
alarms[420](evtEntry:= Tc_Events.AlarmWord27.b4, bEvt:= Alarms_DB.AlarmWord_27.AlarmWord.4, bConfirm:= bConfirm);
alarms[421](evtEntry:= Tc_Events.AlarmWord27.b5, bEvt:= Alarms_DB.AlarmWord_27.AlarmWord.5, bConfirm:= bConfirm);
alarms[422](evtEntry:= Tc_Events.AlarmWord27.b6, bEvt:= Alarms_DB.AlarmWord_27.AlarmWord.6, bConfirm:= bConfirm);
alarms[423](evtEntry:= Tc_Events.AlarmWord27.b7, bEvt:= Alarms_DB.AlarmWord_27.AlarmWord.7, bConfirm:= bConfirm);
alarms[424](evtEntry:= Tc_Events.AlarmWord27.b8, bEvt:= Alarms_DB.AlarmWord_27.AlarmWord.8, bConfirm:= bConfirm);
alarms[425](evtEntry:= Tc_Events.AlarmWord27.b9, bEvt:= Alarms_DB.AlarmWord_27.AlarmWord.9, bConfirm:= bConfirm);
alarms[426](evtEntry:= Tc_Events.AlarmWord27.b10, bEvt:= Alarms_DB.AlarmWord_27.AlarmWord.10, bConfirm:= bConfirm);
alarms[427](evtEntry:= Tc_Events.AlarmWord27.b11, bEvt:= Alarms_DB.AlarmWord_27.AlarmWord.11, bConfirm:= bConfirm);
alarms[428](evtEntry:= Tc_Events.AlarmWord27.b12, bEvt:= Alarms_DB.AlarmWord_27.AlarmWord.12, bConfirm:= bConfirm);
alarms[429](evtEntry:= Tc_Events.AlarmWord27.b13, bEvt:= Alarms_DB.AlarmWord_27.AlarmWord.13, bConfirm:= bConfirm);
alarms[430](evtEntry:= Tc_Events.AlarmWord27.b14, bEvt:= Alarms_DB.AlarmWord_27.AlarmWord.14, bConfirm:= bConfirm);
alarms[431](evtEntry:= Tc_Events.AlarmWord27.b15, bEvt:= Alarms_DB.AlarmWord_27.AlarmWord.15, bConfirm:= bConfirm);
*)

//test
IF GVL.alarm_test THEN
	//i := i+1;
	Alarms_DB.MCP.AlarmWord := 16#FFFF;
	Alarms_DB.Section1.AlarmWord := 16#FFFF;
	Alarms_DB.Section2.AlarmWord := 16#FFFF;
	Alarms_DB.Section3.AlarmWord := 16#FFFF;
	Alarms_DB.Section4.AlarmWord := 16#FFFF;
	Alarms_DB.AlarmWord5.AlarmWord := 16#FFFF;
	Alarms_DB.AlarmWord7.AlarmWord := 16#FFFF;
	//Alarms_DB.Coil3.AlarmWord := 16#FFFF;
	//Alarms_DB.Coil4.AlarmWord := 16#FFFF;
	//Alarms_DB.Coil5.AlarmWord := 16#FFFF;
	//Alarms_DB.Coil6.AlarmWord := 16#FFFF;
	//Alarms_DB.Coil7.AlarmWord := 16#FFFF;
	//Alarms_DB.Coil8.AlarmWord := 16#FFFF;
	//Alarms_DB.Coil9.AlarmWord := 16#FFFF;
	//Alarms_DB.Coil10.AlarmWord := 16#FFFF;
	//Alarms_DB.AlarmWord_11.AlarmWord := 16#FFFF;
	//Alarms_DB.AlarmWord_22.AlarmWord := 16#FFFF;
	//Alarms_DB.AlarmWord_23.AlarmWord := 16#FFFF;
	//Alarms_DB.AlarmWord_24.AlarmWord := 16#FFFF;
	//Alarms_DB.AlarmWord_25.AlarmWord := 16#FFFF;
	//Alarms_DB.AlarmWord_26.AlarmWord := 16#FFFF;
	//Alarms_DB.AlarmWord_27.AlarmWord := 16#FFFF;
END_IF


//Clear Alarm Word
IF bConfirm THEN
	Alarms_DB.MCP.AlarmWord := 0;
	Alarms_DB.Section1.AlarmWord := 0;
	Alarms_DB.Section2.AlarmWord := 0;
	Alarms_DB.Section3.AlarmWord := 0;
	Alarms_DB.Section4.AlarmWord := 0;
	Alarms_DB.AlarmWord5.AlarmWord := 0;
	Alarms_DB.AlarmWord7.AlarmWord := 0;
	(*Alarms_DB.Coil3.AlarmWord := 0;
	Alarms_DB.Coil4.AlarmWord := 0;
	Alarms_DB.Coil5.AlarmWord := 0;
	Alarms_DB.Coil6.AlarmWord := 0;
	Alarms_DB.Coil7.AlarmWord := 0;
	Alarms_DB.Coil8.AlarmWord := 0;
	Alarms_DB.Coil9.AlarmWord := 0;
	Alarms_DB.Coil10.AlarmWord := 0;
	Alarms_DB.AlarmWord_11.AlarmWord := 0;
	Alarms_DB.AlarmWord_22.AlarmWord := 0;
	Alarms_DB.AlarmWord_23.AlarmWord := 0;
	Alarms_DB.AlarmWord_24.AlarmWord := 0;
	Alarms_DB.AlarmWord_25.AlarmWord := 0;
	Alarms_DB.AlarmWord_26.AlarmWord := 0;
	Alarms_DB.AlarmWord_27.AlarmWord := 0;
	*)
END_IF;

END_PROGRAM

// ---- POUs/Sequence.TcPOU
PROGRAM Sequence
VAR
	ePulseState : E_PulseState;
	eCommand	: E_Command;
	eStatus		: E_Status;
	
	ChargeRlyDelayON_Timer  : TON;
	ChargeRlyDelayDONE		: BOOL;
	ChargeRlyDelayON_PT		: TIME := T#250MS; //used for delay close and delay open for safe mode
	AbortPSnRlyDelay_Timer	: TON;
	AbortPSnRlyDelay_PT		: TIME := T#5MS; //defualt is 5ms
	AbortPSnRlyDelayDONE	: BOOL;
	ChargeCompleted			: BOOL;
	ChargingRunOutTMR_TON	: TON;
	ChargingRunOutTMR_ET	: TIME;
	ChargedRunOutTMR_TON	: TON;
	ChargedRunOutTMR_ET		: TIME;
	
	DumpingRunOutTMR_TON 	: TON;
	DumpingRunOutTMR_PT		: TIME := T#180S;
	DumpingRunOutTMR_ET		: TIME;
	LocalDumpActive			: BOOL := FALSE;
	Dump					: Dump_FB;	
	LocalDumpElapse			: REAL;				
		
	ReadyToCharge 			: BOOL;
	StartChargingBroadcast	: BOOL := FALSE;
	StartCharger			: ARRAY[1..8] OF BOOL;
	StartGLS3Charger		: BOOL;
	
	SparkGapCharger_TON		: TON;
	SparkGapCharger_PT		: TIME := T#1S;
	SparkGapCharger_ET		: TIME;
	
	i : INT := 1; // charger 1-8
	j : INT := 1; // section 1 - 3
	k : INT := 1;
	
	ChargeTimeFinished		: BOOL;
END_VAR

//Critical Delay Time
HMI_DB.ChargerHVOFF_rlyDelayPT := INT_TO_TIME(HMI_DB.ChargerHVOFF_rlyDelayPT_INT);
AbortPSnRlyDelay_PT := HMI_DB.ChargerHVOFF_rlyDelayPT;

//hv output delay
HMI_DB.HVONdelayPT := INT_TO_TIME (HMI_DB.HVONdelayPT_INT);
ChargeRlyDelayON_PT := HMI_DB.HVONdelayPT;

//runout timer
HMI_DB.RunOutTMR_PT := INT_TO_TIME (HMI_DB.RunOutTMR_PT_INT*1000);
HMI_DB.RunOutTMR_elapse := (TIME_TO_INT (HMI_DB.RunOutTMR_PT - ChargedRunOutTMR_TON.ET))/1000;
HMI_DB.ChargingRunOutTMR_elapse := TIME_TO_INT(ChargingRunOutTMR_TON.PT/1000 - ChargingRunOutTMR_TON.ET/1000);

//charge realy timer 
ChargeRlyDelayON_Timer(PT := ChargeRlyDelayON_PT);

//screen room asks to go to idle, it will go to safe state. 
//GVL.RemoteModeSelected is MCP_IO.RemoteModeSelected OR HMI_DB.RemoteModeSelected 
IF GVL.RemoteModeSelected = TRUE AND eCommand = E_Command.IDLE AND Trips_DB.NoFaultDetected = TRUE 
	THEN
		ePulseState := E_PulseState.SAFE;
END_IF;
	//at anypoint if screen room wants abort or hmi abort pb is pressed
IF eCommand = E_Command.ABORT OR HMI_DB.AbortPB = TRUE //OR Trips_DB.AnyEstopPressed = TRUE 
	THEN
	 	ePulseState := E_PulseState.ABORT;
END_IF;

IF Trips_DB.NoFaultDetected = FALSE 
	THEN
		ePulseState := E_PulseState.TRIPPED;
END_IF;

IF GVL.RemoteModeSelected = FALSE AND Trips_DB.NoFaultDetected = TRUE 
	THEN
		ePulseState := E_PulseState.LOCALMODE;
END_IF;

//lift machine GND
IF Permissives_DB.AllSectCapsDischarged = FALSE THEN //at least one cap has voltage >10V
	MCP_IO.LiftMachineGND := TRUE;
	ELSE
		MCP_IO.LiftMachineGND := FALSE;
END_IF;

//reset timer
IF ePulseState <> E_PulseState.CHARGING THEN 
	ChargingRunOutTMR_TON (IN := FALSE);
	FOR i := 1 TO 8 BY 1 DO 
		ChargeTime_DB.ChargerDelay_TON[i] (IN := FALSE, PT := ChargeTime_DB.ChargerDelay_PT[i], ET => ChargeTime_DB.ChargerDelay_ET[i]);
		ChargeTime_DB.ChargingTimeElapse_TON[i].IN := FALSE;
		ChargeRlyDelayON_Timer (IN := FALSE);
	END_FOR;
	ChargeTime_DB.PreFormChargeTime_TON (IN := FALSE, PT := ChargeTime_DB.PreFormChargeTime_PT, ET => ChargeTime_DB.PreFormChargeTime_ET);
	ChargeTime_DB.PreFormChargingTimeElapse_TON.IN := FALSE;
END_IF
IF ePulseState <> (E_PulseState.CHARGECOMPLETE OR E_PulseState.DISCONNECTING) THEN 
	ChargedRunOutTMR_TON (IN := FALSE); // only needed in charge complete
END_IF

CASE ePulseState OF 
	
	//Safe OR IDLE
	E_PulseState.SAFE: 
					//TURN OFF ALL CHARGERS
					FOR i := 1 TO 8 BY 1 DO 
						MCP_IO.Charger[i].inhibit := TRUE; // inhibit = high, no output | inhibit = low, allows output
						MCP_IO.Charger[i].HV_ON := FALSE; 
						MCP_IO.Charger[i].voltageSP := 0;
						StartCharger[i] := FALSE; // reset bit
						ChargeTimeFinished := FALSE;
						StartChargingBroadcast := FALSE;
						//reset charger delay timer
						ChargeTime_DB.ChargerDelay_TON[i] (IN := FALSE, PT := ChargeTime_DB.ChargerDelay_PT[i], ET => ChargeTime_DB.ChargerDelay_ET[i]);
						ChargeTime_DB.ChargingTimeElapse_TON[i] (IN := FALSE); 
					END_FOR;
					StartGLS3Charger := FALSE;
					ChargeTime_DB.PreFormChargeTime_TON (IN := FALSE, PT := ChargeTime_DB.PreFormChargeTime_PT, ET => ChargeTime_DB.PreFormChargeTime_ET);
					MCP_IO.GLS1_hvON := FALSE;
					MCP_IO.GLS2_hvON := FALSE;
					MCP_IO.GLS3_hvON := FALSE;
					MCP_IO.GLS1_voltageSP := 0;
					MCP_IO.GLS2_voltageSP := 0;
					MCP_IO.GLS3_voltageSP := 0;
					SparkGapCharger_TON(IN := FALSE);
					//start delay
					IF Permissives_DB.AllChargerHVisON = FALSE THEN 
						ChargeRlyDelayON_Timer (IN := TRUE, PT := ChargeRlyDelayON_PT);	
						ELSE
							ChargeRlyDelayON_Timer (IN := FALSE, PT := ChargeRlyDelayON_PT);				
					END_IF;
					
					IF ChargeRlyDelayON_Timer.Q = TRUE THEN 
						ChargeRlyDelayDONE := TRUE;
						ChargeRlyDelayON_Timer (IN := FALSE);
					END_IF;
					IF ChargeRlyDelayDONE = TRUE THEN
						FOR j := 1 TO 3 BY 1 DO 
							//Open all charge relays after 250ms
							LCP.Section[j].Peak.CloseChargeRelay1 := FALSE; 
							LCP.Section[j].Peak.CloseChargeRelay2 := FALSE; 
							LCP.Section[j].Sust.CloseChargeRelay1 := FALSE;
							LCP.Section[j].Sust.CloseChargeRelay2 := FALSE;
							//close all dump relays  - for SAFE STATE they can all go together
							LCP.Section[j].Peak.OpenDumpRelay1 := FALSE;
							LCP.Section[j].Peak.OpenDumpRelay2 := FALSE;
							LCP.Section[j].Sust.OpenDumpRelay1 := FALSE;
							LCP.Section[j].Sust.OpenDumpRelay2 := FALSE;	
						END_FOR;
						//open all charge rly on form
						LCP.Section[4].Form.CloseChargeRelay1 := FALSE;
						LCP.Section[4].Form.CloseChargeRelay2 := FALSE;
						LCP.Section[4].Form.CloseFormTrigChargeRly := FALSE;
						LCP.Section[4].Form.ClosePreFormChargeRly := FALSE;
						LCP.Section[4].Form.ClosePreFormTrigChargeRly := FALSE;
						//close all dump relay on form
						LCP.Section[4].Form.OpenDumpRelay1 := FALSE;
						LCP.Section[4].Form.OpenDumpRelay2 := FALSE;
						LCP.Section[4].Form.OpenPreFormDumpRly := FALSE;
						LCP.Section[4].Form.OpenFormTrigDumpRly1 := FALSE;
						LCP.Section[4].Form.OpenPreFormTrigDumpRly1 := FALSE;
						
						ChargeRlyDelayDONE := FALSE;
						ChargeRlyDelayON_Timer (IN := FALSE);
					END_IF;
					// short contacts engaged as a permissives to say it is safe???????
					//send status to screen room
					eStatus := E_Status.SAFE;
					
					IF Trips_DB.NoFaultDetected = TRUE AND 
						Permissives_DB.NoShortingUnknowns AND 
						Permissives_DB.AllShortContactEngaged = FALSE
						THEN 
							ReadyToCharge := TRUE;
							ELSE
								ReadyToCharge := FALSE;		
					END_IF;
					//wait for command from screen room
					IF GVL.RemoteModeSelected = TRUE AND ReadyToCharge = TRUE AND eCommand = E_Command.CHARGE 
						THEN
							ePulseState := E_PulseState.CHARGING;
						//ELSIF MCP_IO.RemoteModeSelected = TRUE AND eCommand = E_Command.IDLE THEN
							//ePulseState := E_PulseState.SAFE;
						ELSIF MCP_IO.RemoteModeSelected = TRUE AND eCommand = E_Command.DUMP THEN
							ePulseState := E_PulseState.DUMPING;
					END_IF;
					ChargingRunOutTMR_TON (IN := FALSE);
					ChargedRunOutTMR_TON (IN := FALSE);
					DumpingRunOutTMR_TON (IN := FALSE);
	//Charging
	E_PulseState.CHARGING: 
					MCP_IO.LiftMachineGND := TRUE; //call the bit again in case it did not lift
					
					IF Recipe.PeakSupplyEN = FALSE THEN
						MCP_IO.Charger[1].voltageSP := 0;
						MCP_IO.Charger[2].voltageSP := 0;
						MCP_IO.Charger[3].voltageSP := 0;
					END_IF
					IF Recipe.SustSupplyEN = FALSE THEN
						MCP_IO.Charger[4].voltageSP := 0;
						MCP_IO.Charger[5].voltageSP := 0;
						MCP_IO.Charger[6].voltageSP := 0;
					END_IF
					IF Recipe.FormSupplyEN = FALSE THEN
						MCP_IO.Charger[7].voltageSP := 0;
						MCP_IO.Charger[8].voltageSP := 0;
					END_IF
					IF Recipe.PFormSupplyEN = FALSE THEN
						MCP_IO.GLS3_voltageSP := 0;
					END_IF
					
					//start charging runout timer
					ChargingRunOutTMR_TON (IN := TRUE, PT := (ChargeTime_DB.LongestChargeTime_PT + HMI_DB.RunOutTMR_PT), ET => ChargingRunOutTMR_ET);
	
					//will need the charge time sequence to see stagger each bank's charge time......done
					IF Trips_DB.NoFaultDetected = TRUE THEN 
						FOR j := 1 TO 3 BY 1 DO 
							//Open all dump relays  
							LCP.Section[j].Peak.OpenDumpRelay1 := TRUE;
							LCP.Section[j].Peak.OpenDumpRelay2 := TRUE;
							LCP.Section[j].Sust.OpenDumpRelay1 := TRUE;
							LCP.Section[j].Sust.OpenDumpRelay2 := TRUE;	
						END_FOR;
						//open all dump relay on form
						LCP.Section[4].Form.OpenDumpRelay1 := TRUE;
						LCP.Section[4].Form.OpenDumpRelay2 := TRUE;
						LCP.Section[4].Form.OpenPreFormDumpRly := TRUE;
						LCP.Section[4].Form.OpenFormTrigDumpRly1 := TRUE;
						LCP.Section[4].Form.OpenPreFormTrigDumpRly1 := TRUE;
						//if all dump relays open then close charger relays
						IF Permissives_DB.AllDumpRelaysOpen = TRUE THEN 
							//close all charge rly 
							FOR j := 1 TO 3 BY 1 DO
								IF Recipe.PeakSupplyEN THEN
									LCP.Section[j].Peak.CloseChargeRelay1 := TRUE; 
									LCP.Section[j].Peak.CloseChargeRelay2 := TRUE; 
									ELSE
										LCP.Section[j].Peak.CloseChargeRelay1 := FALSE; 
										LCP.Section[j].Peak.CloseChargeRelay2 := FALSE; 
								END_IF;
								IF Recipe.SustSupplyEN THEN
									LCP.Section[j].Sust.CloseChargeRelay1 := TRUE;
									LCP.Section[j].Sust.CloseChargeRelay2 := TRUE;
									ELSE
										LCP.Section[j].Sust.CloseChargeRelay1 := FALSE;
										LCP.Section[j].Sust.CloseChargeRelay2 := FALSE;
								END_IF
							END_FOR;
							//close all charge rly on form
							IF Recipe.FormSupplyEN THEN
								LCP.Section[4].Form.CloseChargeRelay1 := TRUE;
								LCP.Section[4].Form.CloseChargeRelay2 := TRUE;
								LCP.Section[4].Form.CloseFormTrigChargeRly := TRUE;
								ELSE
									LCP.Section[4].Form.CloseChargeRelay1 := FALSE;
									LCP.Section[4].Form.CloseChargeRelay2 := FALSE;
									LCP.Section[4].Form.CloseFormTrigChargeRly := FALSE;
							END_IF
							
							IF Recipe.PFormSupplyEN THEN
								LCP.Section[4].Form.ClosePreFormChargeRly := TRUE;
								LCP.Section[4].Form.ClosePreFormTrigChargeRly := TRUE;
								ELSE
									LCP.Section[4].Form.ClosePreFormChargeRly := FALSE;
									LCP.Section[4].Form.ClosePreFormTrigChargeRly := FALSE;
							END_IF
						END_IF;	
					END_IF;
					
					IF Trips_DB.NoFaultDetected = TRUE AND Permissives_DB.AllChargeRelaysClosed = TRUE 
						THEN 
							ChargeRlyDelayON_Timer (IN := TRUE, PT := ChargeRlyDelayON_PT);
							ELSE
								ChargeRlyDelayON_Timer (IN := FALSE, PT := ChargeRlyDelayON_PT);
					END_IF;
					//start broadcasting on charger timer
					IF ChargeRlyDelayON_Timer.Q = TRUE THEN 
						StartChargingBroadcast := TRUE;
					END_IF;
					//start timer 
					IF StartChargingBroadcast = TRUE THEN 
						//start total charge time TIMER
						ChargeTime_DB.LongestChargeTime_TON (IN := TRUE, PT := ChargeTime_DB.LongestChargeTime_PT, ET => ChargeTime_DB.LongestChargeTime_ET);
						//Turn inhibit On on all chargers and start timer
						(*FOR i := 1 TO 8 BY 1 DO 
							//MCP_IO.Charger[i].inhibit := TRUE; 
							// delay stagger starts here 
							//ChargeTime_DB.ChargerDelay_TON[i] (IN := TRUE, PT := ChargeTime_DB.ChargerDelay_PT[i], ET => ChargeTime_DB.ChargerDelay_ET[i]);
						END_FOR;*)
						//send voltage SP to chargers
						IF Recipe.PeakSupplyEN = TRUE THEN
							MCP_IO.Charger[1].voltageSP := REAL_TO_DINT (Setpoints.TDKLoad[1].RequiredChargedV * 1000);
							MCP_IO.Charger[2].voltageSP := REAL_TO_DINT (Setpoints.TDKLoad[2].RequiredChargedV * 1000);
							MCP_IO.Charger[3].voltageSP := REAL_TO_DINT (Setpoints.TDKLoad[3].RequiredChargedV * 1000);
							END_IF;
						IF Recipe.SustSupplyEN = TRUE THEN
							MCP_IO.Charger[4].voltageSP := REAL_TO_DINT (Setpoints.TDKLoad[4].RequiredChargedV * 1000);
							MCP_IO.Charger[5].voltageSP := REAL_TO_DINT (Setpoints.TDKLoad[5].RequiredChargedV * 1000);
							MCP_IO.Charger[6].voltageSP := REAL_TO_DINT (Setpoints.TDKLoad[6].RequiredChargedV * 1000);
							END_IF;
						IF Recipe.FormSupplyEN = TRUE THEN
							MCP_IO.Charger[7].voltageSP := REAL_TO_DINT (Setpoints.TDKLoad[7].RequiredChargedV * 1000);
							MCP_IO.Charger[8].voltageSP := REAL_TO_DINT (Setpoints.TDKLoad[8].RequiredChargedV * 1000);
							END_IF;
						IF Recipe.PFormSupplyEN = TRUE THEN
							MCP_IO.GLS3_voltageSP := REAL_TO_DINT (Setpoints.GLSLoad.RequiredChargedV * 1000);
							END_IF
						MCP_IO.GLS1_voltageSP := REAL_TO_DINT (Setpoints.GLS1_VSP * 1000);
						MCP_IO.GLS2_voltageSP := REAL_TO_DINT (Setpoints.GLS2_VSP * 1000);
						
						// delay stagger starts here 
						IF Recipe.PeakSupplyEN = TRUE THEN
							ChargeTime_DB.ChargerDelay_TON[1] (IN := TRUE, PT := ChargeTime_DB.ChargerDelay_PT[1], ET => ChargeTime_DB.ChargerDelay_ET[1]);
							ChargeTime_DB.ChargerDelay_TON[2] (IN := TRUE, PT := ChargeTime_DB.ChargerDelay_PT[2], ET => ChargeTime_DB.ChargerDelay_ET[2]);
							ChargeTime_DB.ChargerDelay_TON[3] (IN := TRUE, PT := ChargeTime_DB.ChargerDelay_PT[3], ET => ChargeTime_DB.ChargerDelay_ET[3]);
						END_IF
						IF Recipe.SustSupplyEN = TRUE THEN
							ChargeTime_DB.ChargerDelay_TON[4] (IN := TRUE, PT := ChargeTime_DB.ChargerDelay_PT[4], ET => ChargeTime_DB.ChargerDelay_ET[4]);
							ChargeTime_DB.ChargerDelay_TON[5] (IN := TRUE, PT := ChargeTime_DB.ChargerDelay_PT[5], ET => ChargeTime_DB.ChargerDelay_ET[5]);
							ChargeTime_DB.ChargerDelay_TON[6] (IN := TRUE, PT := ChargeTime_DB.ChargerDelay_PT[6], ET => ChargeTime_DB.ChargerDelay_ET[6]);
						END_IF
						IF Recipe.FormSupplyEN = TRUE THEN
							ChargeTime_DB.ChargerDelay_TON[7] (IN := TRUE, PT := ChargeTime_DB.ChargerDelay_PT[7], ET => ChargeTime_DB.ChargerDelay_ET[7]);
							ChargeTime_DB.ChargerDelay_TON[8] (IN := TRUE, PT := ChargeTime_DB.ChargerDelay_PT[8], ET => ChargeTime_DB.ChargerDelay_ET[8]);							
						END_IF
						IF Recipe.PFormSupplyEN = TRUE THEN
							ChargeTime_DB.PreFormChargeTime_TON (IN := TRUE, PT := ChargeTime_DB.PreFormChargeTime_PT, ET => ChargeTime_DB.PreFormChargeTime_ET);
						END_IF						
						ChargeRlyDelayON_Timer (IN := FALSE);
						SparkGapCharger_TON(IN := TRUE, PT := (ChargeTime_DB.LongestChargeTime_PT-SparkGapCharger_PT), ET => SparkGapCharger_ET);
					ELSE
						//Turn inhibit High on all chargers and turn off all timer if no broadcasting
						FOR i := 1 TO 8 BY 1 DO 
							MCP_IO.Charger[i].inhibit := TRUE; 
							// turn off timer
							ChargeTime_DB.ChargerDelay_TON[i] (IN := FALSE, PT := ChargeTime_DB.ChargerDelay_PT[i], ET => ChargeTime_DB.ChargerDelay_ET[i]);
						END_FOR;
						ChargeTime_DB.PreFormChargeTime_TON (IN := FALSE, PT := ChargeTime_DB.PreFormChargeTime_PT, ET => ChargeTime_DB.PreFormChargeTime_ET);	
						ChargeTime_DB.LongestChargeTime_TON (IN := FALSE); //reset timer	
						SparkGapCharger_TON(IN := TRUE);						
					END_IF;
					
					//turn on HV output to load	
					IF Recipe.PeakSupplyEN = TRUE AND ChargeTime_DB.ChargerDelay_TON[1].Q = TRUE THEN
						StartCharger[1] := TRUE;
					END_IF
					IF Recipe.PeakSupplyEN = TRUE AND ChargeTime_DB.ChargerDelay_TON[2].Q = TRUE THEN
						StartCharger[2] := TRUE;
					END_IF
					IF Recipe.PeakSupplyEN = TRUE AND ChargeTime_DB.ChargerDelay_TON[3].Q = TRUE THEN
						StartCharger[3] := TRUE;
					END_IF
					IF Recipe.SustSupplyEN = TRUE AND ChargeTime_DB.ChargerDelay_TON[4].Q = TRUE THEN
						StartCharger[4] := TRUE;
					END_IF
					IF Recipe.SustSupplyEN = TRUE AND ChargeTime_DB.ChargerDelay_TON[5].Q = TRUE THEN
						StartCharger[5] := TRUE;
					END_IF
					IF Recipe.SustSupplyEN = TRUE AND ChargeTime_DB.ChargerDelay_TON[6].Q = TRUE THEN
						StartCharger[6] := TRUE;
					END_IF
					IF Recipe.FormSupplyEN = TRUE AND ChargeTime_DB.ChargerDelay_TON[7].Q = TRUE THEN
						StartCharger[7] := TRUE;
					END_IF
					IF Recipe.FormSupplyEN = TRUE AND ChargeTime_DB.ChargerDelay_TON[8].Q = TRUE THEN
						StartCharger[8] := TRUE;
					END_IF

					
					FOR k := 1 TO 8 BY 1 DO

						(*IF ChargeTime_DB.ChargerDelay_TON[k].Q = TRUE THEN
							StartCharger[k] := TRUE;
						END_IF;
						*)
						IF StartCharger[k] = TRUE THEN
							MCP_IO.Charger[k].HV_ON := TRUE; 
							MCP_IO.Charger[k].inhibit := FALSE;
							ChargeTime_DB.ChargerDelay_TON[k] (IN := FALSE, PT := ChargeTime_DB.ChargerDelay_PT[k], ET => ChargeTime_DB.ChargerDelay_ET[k]);
							//start time elapse
							ChargeTime_DB.ChargingTimeElapse_TON[k] (IN := TRUE, PT := REAL_TO_TIME (1000*MCP_IO.Charger[k].ChargeTime.timeToChargeLoad));
						END_IF;
						
						IF ChargeTime_DB.ChargingTimeElapse_TON[k].Q THEN
							StartCharger[k] := FALSE;
							ChargeTime_DB.ChargingTimeElapse_TON[k] (IN := FALSE); 
						END_IF;
					END_FOR
					//GLS 3
					IF ChargeTime_DB.PreFormChargeTime_TON.Q = TRUE AND Recipe.PFormSupplyEN = TRUE THEN
						StartGLS3Charger := TRUE;
					END_IF;
					IF StartGLS3Charger = TRUE THEN 
						MCP_IO.GLS3_hvON := TRUE;
						ChargeTime_DB.PreFormChargeTime_TON (IN := FALSE, PT := ChargeTime_DB.PreFormChargeTime_PT, ET => ChargeTime_DB.PreFormChargeTime_ET);
						//for hmi
						ChargeTime_DB.PreFormChargingTimeElapse_TON (IN := TRUE, PT :=  REAL_TO_TIME (1000*MCP_IO.GLS3_Load.timeToChargeLoad));
					END_IF;
					
					IF ChargeTime_DB.PreFormChargingTimeElapse_TON.Q = TRUE THEN
						StartGLS3Charger := FALSE;
						ChargeTime_DB.PreFormChargingTimeElapse_TON (IN := FALSE);
					END_IF
					
					IF SparkGapCharger_TON.Q = TRUE THEN 
						MCP_IO.GLS1_hvON := TRUE; //turn on spark gap charger
						MCP_IO.GLS2_hvON := TRUE;
						SparkGapCharger_TON(IN := FALSE);
					END_IF
					//turn off inhibit when HV is on
					(*IF Permissives_DB.AllChargerHVisON = TRUE THEN
						FOR i := 1 TO 8 BY 1 DO 
							MCP_IO.Charger[i].inhibit := FALSE; //start current output
						END_FOR;
						//StartChargingBroadcast := FALSE; // reset the broadcast bit whne all chargers 
					END_IF*)
					IF ChargingRunOutTMR_TON.Q = TRUE THEN
						Trips_DB.ChargingTimerRunout := TRUE;
						ChargingRunOutTMR_TON (IN := FALSE);
					END_IF
					
					IF Trips_DB.AnyLossHVONsignal = TRUE OR Trips_DB.ChargingTimerRunout = TRUE THEN 
						StartChargingBroadcast := FALSE; // reset the broadcast bit whne all chargers
						ChargeTimeFinished := FALSE; //reset chargetime done bit
						ChargingRunOutTMR_TON (IN := FALSE);
						FOR i := 1 TO 8 BY 1 DO 
							ChargeTime_DB.ChargingTimeElapse_TON[i] (IN := FALSE);							
						END_FOR
						ChargeTime_DB.PreFormChargingTimeElapse_TON (IN := FALSE);
						ePulseState := E_PulseState.TRIPPED; 
					END_IF
					//send status to screen room
					eStatus := E_Status.CHARGING;
					
					IF ChargeTime_DB.LongestChargeTime_TON.Q = TRUE THEN 
						ChargeTimeFinished := TRUE;
						ChargeTime_DB.LongestChargeTime_TON (IN := FALSE); //reset timer
					END_IF
					
					IF ChargeTimeFinished = TRUE THEN 
						//reset elapse timer
						FOR i := 1 TO 8 BY 1 DO 
							StartCharger[i] := FALSE;
							ChargeTime_DB.ChargingTimeElapse_TON[i] (IN := FALSE);							
						END_FOR
						ChargeTime_DB.PreFormChargingTimeElapse_TON (IN := FALSE);
						StartGLS3Charger := FALSE;
						MCP_IO.GLS1_hvON := FALSE; //turn off spark gap charger
						MCP_IO.GLS2_hvON := FALSE;
						SparkGapCharger_TON(IN := FALSE);
					END_IF
					//condition for charge complete
					IF Permissives_DB.AllChargerEOC = TRUE AND ChargeTimeFinished = TRUE AND Permissives_DB.AllSectCapsFullyCharged = TRUE THEN 
						ChargeCompleted := TRUE;
						ELSE
							ChargeCompleted := FALSE;
					END_IF
					
					//if cap voltage feedback >= charger setpoints && EOC && all timer runout then chargecomplete
					IF ChargeCompleted = TRUE THEN 
						FOR i := 1 TO 8 BY 1 DO 
							MCP_IO.Charger[i].HV_ON := FALSE; 
							MCP_IO.Charger[i].inhibit := TRUE;
							StartCharger[i] := FALSE;
							ChargeTime_DB.ChargingTimeElapse_TON[i] (IN := FALSE);	
							//ChargeTime_DB.ChargerDelay_TON[i] (IN := FALSE, PT := ChargeTime_DB.ChargerDelay_PT[i], ET => ChargeTime_DB.ChargerDelay_ET[i]);
						END_FOR;
						StartGLS3Charger := FALSE;
						ChargeTime_DB.PreFormChargeTime_TON (IN := FALSE, PT := ChargeTime_DB.PreFormChargeTime_PT, ET => ChargeTime_DB.PreFormChargeTime_ET);
						StartChargingBroadcast := FALSE; // reset the broadcast bit whne all chargers 
						ChargeTimeFinished := FALSE; //reset chargetime done bit
						ePulseState := E_PulseState.CHARGECOMPLETE;
					END_IF
	//Charge complete
	E_PulseState.CHARGECOMPLETE: 
	
					ChargeCompleted := FALSE; //reset bit
					ChargingRunOutTMR_TON (IN := FALSE);
					eStatus := E_Status.CHARGECOMPLETE;
					
					MCP_IO.GLS1_hvON := FALSE; //turn off spark gap charger
					MCP_IO.GLS2_hvON := FALSE;	
					SparkGapCharger_TON(IN := FALSE, PT := SparkGapCharger_PT, ET => SparkGapCharger_ET);
					//start run out timer
					ChargedRunOutTMR_TON (IN := TRUE, PT := HMI_DB.RunOutTMR_PT);
					
					IF ChargedRunOutTMR_TON.Q = TRUE THEN
						Trips_DB.ChargedTimerRunout := TRUE;
						ChargedRunOutTMR_TON (IN := FALSE, PT := HMI_DB.RunOutTMR_PT);
						ePulseState := E_PulseState.DUMPING;
					END_IF
					//turn off charger HV and inhibit 
					FOR i := 1 TO 8 BY 1 DO 
						MCP_IO.Charger[i].inhibit := TRUE;
						MCP_IO.Charger[i].HV_ON := FALSE; 
						ChargeTime_DB.ChargerDelay_TON[i] (IN := FALSE, PT := ChargeTime_DB.ChargerDelay_PT[i], ET => ChargeTime_DB.ChargerDelay_ET[i]);
					END_FOR
					MCP_IO.GLS3_hvON := FALSE;
					ChargeTime_DB.PreFormChargeTime_TON(IN := FALSE);
					
					IF eCommand = E_Command.DISCONNECT THEN 
						ePulseState := E_PulseState.DISCONNECTING;
					END_IF

	//Disconnecting
	E_PulseState.DISCONNECTING:
					eStatus := E_Status.DISCONNECTING;
					//setpoints to 0
					FOR i := 1 TO 8 BY 1 DO
						MCP_IO.Charger[i].voltageSP := 0;
					END_FOR;
					MCP_IO.GLS3_voltageSP := 0;
					//spark gap chargers now turns off
					MCP_IO.GLS1_hvON := FALSE; 
					MCP_IO.GLS2_hvON := FALSE;
					MCP_IO.GLS1_voltageSP := 0;
					MCP_IO.GLS2_voltageSP := 0;
					
					//start run out timer
					ChargedRunOutTMR_TON (IN := TRUE, PT := HMI_DB.RunOutTMR_PT);
					
					IF ChargedRunOutTMR_TON.Q = TRUE THEN
						Trips_DB.ChargedTimerRunout := TRUE;
						ChargedRunOutTMR_TON (IN := FALSE, PT := HMI_DB.RunOutTMR_PT);
						ePulseState := E_PulseState.DUMPING;
					END_IF
					//keep dump relays open, 
					FOR j := 1 TO 3 BY 1 DO 
						//close all dump relays
						LCP.Section[j].Peak.OpenDumpRelay1 := TRUE;
						LCP.Section[j].Peak.OpenDumpRelay2 := TRUE;
						LCP.Section[j].Sust.OpenDumpRelay1 := TRUE;
						LCP.Section[j].Sust.OpenDumpRelay2 := TRUE;	
						//Open all charge relays
						LCP.Section[j].Peak.CloseChargeRelay1 := FALSE; 
						LCP.Section[j].Peak.CloseChargeRelay2 := FALSE; 
						LCP.Section[j].Sust.CloseChargeRelay1 := FALSE;
						LCP.Section[j].Sust.CloseChargeRelay2 := FALSE;
					END_FOR;	
					//close all dump relay on form
					LCP.Section[4].Form.OpenDumpRelay1 := TRUE;
					LCP.Section[4].Form.OpenDumpRelay2 := TRUE;
					LCP.Section[4].Form.OpenPreFormDumpRly := TRUE;
					LCP.Section[4].Form.OpenFormTrigDumpRly1 := TRUE;
					LCP.Section[4].Form.OpenPreFormTrigDumpRly1 := TRUE;

					//open all charge rly on form
					LCP.Section[4].Form.CloseChargeRelay1 := FALSE;
					LCP.Section[4].Form.CloseChargeRelay2 := FALSE;
					LCP.Section[4].Form.CloseFormTrigChargeRly := FALSE;
					LCP.Section[4].Form.ClosePreFormChargeRly := FALSE;
					LCP.Section[4].Form.ClosePreFormTrigChargeRly := FALSE;	
					
					IF Permissives_DB.AllChargeRelaysClosed = FALSE AND Permissives_DB.AllDumpRelaysOpen THEN
						eStatus := E_Status.DISCONNECTED; //send status to main plc
					END_IF;
					
					IF eCommand = E_Command.ABORT THEN 
						ePulseState := E_PulseState.ABORT;
					ELSIF eCommand = E_Command.DUMP THEN
						ePulseState := E_PulseState.DUMPING;
					END_IF;
	//Dumping
	E_PulseState.DUMPING:  
					//start dump runout timer
					DumpingRunOutTMR_TON (IN := TRUE, PT := DumpingRunOutTMR_PT, ET => DumpingRunOutTMR_ET);
					
					IF DumpingRunOutTMR_TON.Q = TRUE THEN //if timer run out, and in remoter mode go to trip
						Trips_DB.DumpTimerRunout := TRUE;
						DumpingRunOutTMR_TON (IN := FALSE);
						ePulseState := E_PulseState.TRIPPED;
					END_IF
					
					//TURN OFF ALL CHARGERS
					FOR i := 1 TO 8 BY 1 DO 
						MCP_IO.Charger[i].inhibit := TRUE; 		
						MCP_IO.Charger[i].HV_ON := FALSE; 
						MCP_IO.Charger[i].voltageSP := 0;
			
						ChargeTime_DB.ChargingTimeElapse_TON[i] (IN := FALSE); //reset charging time elapse
					END_FOR;
					MCP_IO.GLS1_hvON := FALSE;
					MCP_IO.GLS2_hvON := FALSE;
					MCP_IO.GLS3_hvON := FALSE;
					MCP_IO.GLS1_voltageSP := 0;
					MCP_IO.GLS2_voltageSP := 0;
					MCP_IO.GLS3_voltageSP := 0;
					
					ChargeTime_DB.PreFormChargingTimeElapse_TON (IN := FALSE);
					//start delay
					AbortPSnRlyDelay_Timer (IN := TRUE, PT := AbortPSnRlyDelay_PT);					
					
					IF AbortPSnRlyDelay_Timer.Q = TRUE THEN 
						AbortPSnRlyDelayDONE := TRUE;
						AbortPSnRlyDelay_Timer (IN := FALSE);
					END_IF;
					
					IF 	AbortPSnRlyDelayDONE = TRUE THEN
						FOR j := 1 TO 3 BY 1 DO 
							//Open all charge relays
							LCP.Section[j].Peak.CloseChargeRelay1 := FALSE; 
							LCP.Section[j].Peak.CloseChargeRelay2 := FALSE; 
							LCP.Section[j].Sust.CloseChargeRelay1 := FALSE;
							LCP.Section[j].Sust.CloseChargeRelay2 := FALSE;
							//close all dump relays  - for SAFE STATE they can all go together
							LCP.Section[j].Peak.OpenDumpRelay1 := FALSE;
							LCP.Section[j].Peak.OpenDumpRelay2 := FALSE;
							LCP.Section[j].Sust.OpenDumpRelay1 := FALSE;
							LCP.Section[j].Sust.OpenDumpRelay2 := FALSE;	
						END_FOR;
						//open all charge rly on form
						LCP.Section[4].Form.CloseChargeRelay1 := FALSE;
						LCP.Section[4].Form.CloseChargeRelay2 := FALSE;
						LCP.Section[4].Form.CloseFormTrigChargeRly := FALSE;
						LCP.Section[4].Form.ClosePreFormChargeRly := FALSE;
						LCP.Section[4].Form.ClosePreFormTrigChargeRly := FALSE;
						//close all dump relay on form
						LCP.Section[4].Form.OpenDumpRelay1 := FALSE;
						LCP.Section[4].Form.OpenDumpRelay2 := FALSE;
						LCP.Section[4].Form.OpenPreFormDumpRly := FALSE;
						LCP.Section[4].Form.OpenFormTrigDumpRly1 := FALSE;
						LCP.Section[4].Form.OpenPreFormTrigDumpRly1 := FALSE;
						
						AbortPSnRlyDelay_Timer (IN := FALSE);
						AbortPSnRlyDelayDONE := FALSE;
					END_IF;
					
					eStatus := E_Status.DUMPING;
					
					IF (Permissives_DB.AllSectCapsDischarged = TRUE AND 
						Permissives_DB.AllDumpRelaysOpen = FALSE AND 
						eCommand = E_Command.IDLE AND 
						GVL.RemoteModeSelected = TRUE) 
						THEN 
							ePulseState := E_PulseState.SAFE;
					END_IF
	
	//Abort
	E_PulseState.ABORT: 
					//do something
					//ChargingRunOutTMR_TON (IN := FALSE);
					//TURN OFF ALL CHARGERS' outputs
					FOR i := 1 TO 8 BY 1 DO 
						MCP_IO.Charger[i].inhibit := TRUE; //active low
						MCP_IO.Charger[i].HV_ON := FALSE; 
						MCP_IO.Charger[i].voltageSP := 0;
						
						ChargeTime_DB.ChargingTimeElapse_TON[i] (IN := FALSE);  
					END_FOR;
					MCP_IO.GLS1_hvON := FALSE;
					MCP_IO.GLS2_hvON := FALSE;
					MCP_IO.GLS3_hvON := FALSE;
					
					MCP_IO.GLS1_voltageSP := 0;
					MCP_IO.GLS2_voltageSP := 0;
					MCP_IO.GLS3_voltageSP := 0;
					//start delay
					AbortPSnRlyDelay_Timer (IN := TRUE, PT := AbortPSnRlyDelay_PT);					
					
					IF AbortPSnRlyDelay_Timer.Q = TRUE THEN 
						AbortPSnRlyDelayDONE := TRUE;
						AbortPSnRlyDelay_Timer (IN := FALSE);
					END_IF;
					IF AbortPSnRlyDelayDONE = TRUE THEN
						FOR j := 1 TO 3 BY 1 DO 
							//Open all charge relays
							LCP.Section[j].Peak.CloseChargeRelay1 := FALSE; 
							LCP.Section[j].Peak.CloseChargeRelay2 := FALSE; 
							LCP.Section[j].Sust.CloseChargeRelay1 := FALSE;
							LCP.Section[j].Sust.CloseChargeRelay2 := FALSE;
							//close all dump relays  - for SAFE STATE they can all go together
							LCP.Section[j].Peak.OpenDumpRelay1 := FALSE;
							LCP.Section[j].Peak.OpenDumpRelay2 := FALSE;
							LCP.Section[j].Sust.OpenDumpRelay1 := FALSE;
							LCP.Section[j].Sust.OpenDumpRelay2 := FALSE;	
						END_FOR;
						//open all charge rly on form
						LCP.Section[4].Form.CloseChargeRelay1 := FALSE;
						LCP.Section[4].Form.CloseChargeRelay2 := FALSE;
						LCP.Section[4].Form.CloseFormTrigChargeRly := FALSE;
						LCP.Section[4].Form.ClosePreFormChargeRly := FALSE;
						LCP.Section[4].Form.ClosePreFormTrigChargeRly := FALSE;
						//close all dump relay on form
						LCP.Section[4].Form.OpenDumpRelay1 := FALSE;
						LCP.Section[4].Form.OpenDumpRelay2 := FALSE;
						LCP.Section[4].Form.OpenPreFormDumpRly := FALSE;
						LCP.Section[4].Form.OpenFormTrigDumpRly1 := FALSE;
						LCP.Section[4].Form.OpenPreFormTrigDumpRly1 := FALSE;
						
						AbortPSnRlyDelay_Timer (IN := FALSE);
						AbortPSnRlyDelayDONE := FALSE;		
					END_IF;
	
					eStatus := E_Status.ABORT;
					//logic to go back to safe state.
					IF (Trips_DB.NoFaultDetected = TRUE AND 
						Permissives_DB.AllDumpRelaysOpen = FALSE AND 
						Permissives_DB.AllChargeRelaysClosed = FALSE AND
						Permissives_DB.AllChargerHVisON = FALSE) OR (eCommand = E_Command.IDLE AND MCP_IO.RemoteModeSelected = TRUE)
						THEN 
							AbortPSnRlyDelayDONE := FALSE;
							ePulseState := E_PulseState.SAFE;	
					END_IF;
					
	//Abort
	E_PulseState.TRIPPED: 
					eStatus := E_Status.TRIPPED;
					//reset dumping run out timer
					DumpingRunOutTMR_TON (IN := FALSE, PT := DumpingRunOutTMR_PT, ET => DumpingRunOutTMR_ET);
					
					FOR i := 1 TO 8 BY 1 DO 
						MCP_IO.Charger[i].inhibit := TRUE; //active low
						MCP_IO.Charger[i].HV_ON := FALSE; 
					END_FOR;
					
					FOR j := 1 TO 3 BY 1 DO 
						//close all dump relays
						LCP.Section[j].Peak.OpenDumpRelay1 := FALSE;
						LCP.Section[j].Peak.OpenDumpRelay2 := FALSE;
						LCP.Section[j].Sust.OpenDumpRelay1 := FALSE;
						LCP.Section[j].Sust.OpenDumpRelay2 := FALSE;
						//Open all charge relays
						LCP.Section[j].Peak.CloseChargeRelay1 := FALSE; 
						LCP.Section[j].Peak.CloseChargeRelay2 := FALSE; 
						LCP.Section[j].Sust.CloseChargeRelay1 := FALSE;
						LCP.Section[j].Sust.CloseChargeRelay2 := FALSE;	
					END_FOR;	
					//close all dump relay on form
					LCP.Section[4].Form.OpenDumpRelay1 := FALSE;
					LCP.Section[4].Form.OpenDumpRelay2 := FALSE;
					LCP.Section[4].Form.OpenPreFormDumpRly := FALSE;
					LCP.Section[4].Form.OpenFormTrigDumpRly1 := FALSE;
					LCP.Section[4].Form.OpenPreFormTrigDumpRly1 := FALSE;
			
					//open all charge rly on form
					LCP.Section[4].Form.CloseChargeRelay1 := FALSE;
					LCP.Section[4].Form.CloseChargeRelay2 := FALSE;
					LCP.Section[4].Form.CloseFormTrigChargeRly := FALSE;
					LCP.Section[4].Form.ClosePreFormChargeRly := FALSE;
					LCP.Section[4].Form.ClosePreFormTrigChargeRly := FALSE;	
	
					FOR i := 1 TO 8 BY 1 DO
						MCP_IO.Charger[i].voltageSP := 0;
						ChargeTime_DB.ChargingTimeElapse_TON[i] (IN := FALSE);  
					END_FOR;					
					MCP_IO.GLS1_hvON := FALSE;
					MCP_IO.GLS2_hvON := FALSE;
					MCP_IO.GLS3_hvON := FALSE;
					
					MCP_IO.GLS1_voltageSP := 0;
					MCP_IO.GLS2_voltageSP := 0;
					MCP_IO.GLS3_voltageSP := 0;
									
					//ChargingRunOutTMR_TON (IN := FALSE);
					//logic to go back to safe state.
					IF (Trips_DB.NoFaultDetected = TRUE OR HMI_DB.NoFaultDetectedBP = TRUE) AND 
						(Permissives_DB.AllDumpRelaysOpen = FALSE OR HMI_DB.AllDumpRelaysOpenBP = TRUE) AND 
						(Permissives_DB.AllChargeRelaysClosed = FALSE OR HMI_DB.AllChargeRelayCloseBP = TRUE) AND
						Permissives_DB.AllChargerHVisON = FALSE  AND
						(Permissives_DB.SafetyOK = TRUE OR HMI_DB.SafetyOKBP = TRUE)
						THEN 
							ePulseState := E_PulseState.SAFE;	
					END_IF;
	//lOCAL MODE
	E_PulseState.LOCALMODE:
					eStatus := E_Status.LOCAL_MODE;
					
					IF HMI_DB.DumpALLPB_Local = TRUE THEN
						LocalDumpActive := TRUE;
					END_IF
					
					//Local dump activated			
					IF LocalDumpActive = TRUE THEN 
						//reset all HMI Switches
						HMI_DB.OpenAllDumpRlyPB := FALSE;
						HMI_DB.CloseAllChargeRlyPB := FALSE;
						
						HMI_DB.CloseAllPeakChargRlySW := FALSE;
						HMI_DB.CloseAllSustChargRlySW := FALSE;
						HMI_DB.CloseAllFormChargRlySW := FALSE;
						HMI_DB.CloseAllPreFormChargRlySW := FALSE;
						HMI_DB.ClosePreFormTrigChargeRlySW := FALSE;
						HMI_DB.CloseFormTrigChargeRlySW := FALSE;
						
						HMI_DB.OpenAllPeakDumpRlySW := FALSE;
						HMI_DB.OpenAllSustDumpRlySW := FALSE;
						HMI_DB.OpenAllFormDumpRlySW := FALSE;
						HMI_DB.OpenAllPreFormDumpRlySW := FALSE;
						HMI_DB.OpenPreFormTrigDumpRlySW := FALSE;
						HMI_DB.OpenFormTrigDumpRlySW := FALSE;
						
						HMI_DB.PeakHVONsw := FALSE;
						HMI_DB.SustHVONsw := FALSE;
						HMI_DB.FormHVONsw := FALSE;
						HMI_DB.PreFormHVONsw := FALSE;
						HMI_DB.GLS1HVONsw := FALSE;
						HMI_DB.GLS2HVONsw := FALSE;			
						
						Dump( EN := TRUE, IN1 := Permissives_DB.AllSectCapsDischarged, IN2 := Permissives_DB.AllDumpRelaysOpen);
						DumpingRunOutTMR_TON (IN := TRUE, PT := DumpingRunOutTMR_PT, ET => DumpingRunOutTMR_ET);
						LocalDumpElapse := Dump.DumpingRunOut_Elapse;
						ELSE 
							Dump.EN := FALSE; 
							DumpingRunOutTMR_TON (IN := FALSE);
					END_IF;
					
					IF DumpingRunOutTMR_TON.Q = TRUE THEN 
						Trips_DB.DumpTimerRunout := TRUE;
						DumpingRunOutTMR_TON (IN := FALSE);
					END_IF
					
					IF Trips_DB.DumpTimerRunout = TRUE THEN
						ePulseState := E_PulseState.TRIPPED;
					END_IF

